LIN {X 0,Y 309.388,Z 528.778,A -85,B 0,C 180,E1 -16861.301,E2 -16861.301} C_VEL
LIN {X 0,Y 303.998,Z 522.37,A -85,B 0,C 180,E1 -16862.326,E2 -16862.326} C_VEL
LIN {X 0,Y 299.975,Z 517.415,A -85,B 0,C 180,E1 -16863.035,E2 -16863.035} C_VEL
LIN {X 0,Y 294.271,Z 509.19,A -85,B 0,C 180,E1 -16864.039,E2 -16864.039} C_VEL
LIN {X 0,Y 291.63,Z 504.474,A -85,B 0,C 180,E1 -16864.56,E2 -16864.56} C_VEL
LIN {X 0,Y 291.395,Z 503.436,A -85,B 0,C 180,E1 -16864.862,E2 -16864.862} C_VEL
LIN {X 0,Y 291.393,Z 503.278,A -85,B 0,C 180,E1 -16867.26,E2 -16867.26} C_VEL
LIN {X 0,Y 291.4,Z 503.295,A -85,B 0,C 180,E1 -16870.63,E2 -16870.63} C_VEL
LIN {X 0,Y 291.4,Z 503.269,A -85,B 0,C 180,E1 -16874.379,E2 -16874.379} C_VEL
LIN {X 0,Y 291.383,Z 503.302,A -85,B 0,C 180,E1 -16878.39,E2 -16878.39} C_VEL
LIN {X 0,Y 291.377,Z 503.316,A -85,B 0,C 180,E1 -16881.163,E2 -16881.163} C_VEL
LIN {X 0,Y 291.378,Z 503.299,A -85,B 0,C 180,E1 -16884.629,E2 -16884.629} C_VEL
LIN {X 0,Y 291.368,Z 503.305,A -85,B 0,C 180,E1 -16887.951,E2 -16887.951} C_VEL
LIN {X 0,Y 291.376,Z 503.307,A -85,B 0,C 180,E1 -16891.159,E2 -16891.159} C_VEL
LIN {X 0,Y 291.409,Z 503.295,A -85,B 0,C 180,E1 -16894.272,E2 -16894.272} C_VEL
LIN {X 0,Y 291.374,Z 503.303,A -85,B 0,C 180,E1 -16897.3,E2 -16897.3} C_VEL
LIN {X 0,Y 291.451,Z 503.298,A -85,B 0,C 180,E1 -16900.27,E2 -16900.27} C_VEL
LIN {X 0,Y 291.534,Z 503.284,A -85,B 0,C 180,E1 -16904.635,E2 -16904.635} C_VEL
LIN {X 0,Y 291.528,Z 503.272,A -85,B 0,C 180,E1 -16908.881,E2 -16908.881} C_VEL
LIN {X 0,Y 291.681,Z 503.258,A -85,B 0,C 180,E1 -16911.688,E2 -16911.688} C_VEL
LIN {X 0,Y 291.623,Z 503.281,A -85,B 0,C 180,E1 -16914.469,E2 -16914.469} C_VEL
LIN {X 0,Y 291.883,Z 503.219,A -85,B 0,C 180,E1 -16918.621,E2 -16918.621} C_VEL
LIN {X 0,Y 291.883,Z 503.248,A -85,B 0,C 180,E1 -16921.38,E2 -16921.38} C_VEL
LIN {X 0,Y 291.736,Z 503.243,A -85,B 0,C 180,E1 -16926.919,E2 -16926.919} C_VEL
LIN {X 0,Y 291.623,Z 503.283,A -85,B 0,C 180,E1 -16929.713,E2 -16929.713} C_VEL
LIN {X 0,Y 291.511,Z 503.266,A -85,B 0,C 180,E1 -16933.881,E2 -16933.881} C_VEL
LIN {X 0,Y 290.876,Z 503.358,A -85,B 0,C 180,E1 -16935.034,E2 -16935.034} C_VEL
LIN {X 0,Y 287.966,Z 503.74,A -85,B 0,C 180,E1 -16936.908,E2 -16936.908} C_VEL
LIN {X 0,Y 285.486,Z 504.04,A -85,B 0,C 180,E1 -16938.43,E2 -16938.43} C_VEL
LIN {X 0,Y 284.448,Z 504.156,A -85,B 0,C 180,E1 -16939.612,E2 -16939.612} C_VEL
LIN {X 0,Y 284.379,Z 504.161,A -85,B 0,C 180,E1 -16940.012,E2 -16940.012} C_VEL
LIN {X 0,Y 284.33,Z 504.191,A -85,B 0,C 180,E1 -16943.86,E2 -16943.86} C_VEL
LIN {X 0,Y 284.388,Z 504.161,A -85,B 0,C 180,E1 -16947.172,E2 -16947.172} C_VEL
LIN {X 0,Y 284.29,Z 504.193,A -85,B 0,C 180,E1 -16951.276,E2 -16951.276} C_VEL
LIN {X 0,Y 284.359,Z 504.19,A -85,B 0,C 180,E1 -16955.355,E2 -16955.355} C_VEL
LIN {X 0,Y 284.327,Z 504.179,A -85,B 0,C 180,E1 -16958.167,E2 -16958.167} C_VEL
LIN {X 0,Y 284.3,Z 504.187,A -85,B 0,C 180,E1 -16961.871,E2 -16961.871} C_VEL
LIN {X 0,Y 284.253,Z 504.171,A -85,B 0,C 180,E1 -16966.19,E2 -16966.19} C_VEL
LIN {X 0,Y 284.335,Z 504.299,A -85,B 0,C 180,E1 -16968.964,E2 -16968.964} C_VEL
LIN {X 0,Y 286.321,Z 512.531,A -85,B 0,C 180,E1 -16972.592,E2 -16972.592} C_VEL
LIN {X 0,Y 287.571,Z 518.102,A -85,B 0,C 180,E1 -16974.858,E2 -16974.858} C_VEL
LIN {X 0,Y 290.631,Z 524.68,A -85,B 0,C 180,E1 -16975.534,E2 -16975.534} C_VEL
LIN {X 0,Y 297.502,Z 539.552,A -85,B 0,C 180,E1 -16976.851,E2 -16976.851} C_VEL
LIN {X 0,Y 300.601,Z 547.16,A -85,B 0,C 180,E1 -16977.444,E2 -16977.444} C_VEL
LIN {X 0,Y 304.86,Z 568.834,A -85,B 0,C 180,E1 -16978.537,E2 -16978.537} C_VEL
LIN {X 0,Y 305.547,Z 572.651,A -85,B 0,C 180,E1 -16978.718,E2 -16978.718} C_VEL
LIN {X 0,Y 302.81,Z 652.99,A -85,B 0,C 180,E1 -16980.599,E2 -16980.599} C_VEL
LIN {X 0,Y 302.066,Z 664.113,A -85,B 0,C 180,E1 -16980.991,E2 -16980.991} C_VEL
LIN {X 0,Y 301.043,Z 674.654,A -85,B 0,C 180,E1 -16981.503,E2 -16981.503} C_VEL
LIN {X 0,Y 299.622,Z 685.804,A -85,B 0,C 180,E1 -16982.213,E2 -16982.213} C_VEL
LIN {X 0,Y 298.202,Z 695.774,A -85,B 0,C 180,E1 -16983.021,E2 -16983.021} C_VEL
LIN {X 0,Y 296.541,Z 705.698,A -85,B 0,C 180,E1 -16983.996,E2 -16983.996} C_VEL
LIN {X 0,Y 294.822,Z 715.628,A -85,B 0,C 180,E1 -16985.189,E2 -16985.189} C_VEL
LIN {X 0,Y 292.991,Z 724.837,A -85,B 0,C 180,E1 -16986.498,E2 -16986.498} C_VEL
LIN {X 0,Y 290.978,Z 733.855,A -85,B 0,C 180,E1 -16988.015,E2 -16988.015} C_VEL
LIN {X 0,Y 289.468,Z 740.831,A -85,B 0,C 180,E1 -16989.388,E2 -16989.388} C_VEL
LIN {X 0,Y 287.783,Z 748.355,A -85,B 0,C 180,E1 -16991.121,E2 -16991.121} C_VEL
LIN {X 0,Y 286.364,Z 754.83,A -85,B 0,C 180,E1 -16992.872,E2 -16992.872} C_VEL
LIN {X 0,Y 285.058,Z 761.375,A -85,B 0,C 180,E1 -16994.997,E2 -16994.997} C_VEL
LIN {X 0,Y 283.97,Z 766.81,A -85,B 0,C 180,E1 -16997.13,E2 -16997.13} C_VEL
LIN {X 0,Y 283.149,Z 771.256,A -85,B 0,C 180,E1 -16999.272,E2 -16999.272} C_VEL
LIN {X 0,Y 282.689,Z 774.805,A -85,B 0,C 180,E1 -17001.422,E2 -17001.422} C_VEL
LIN {X 0,Y 282.492,Z 776.748,A -85,B 0,C 180,E1 -17002.854,E2 -17002.854} C_VEL
LIN {X 0,Y 282.301,Z 779.436,A -85,B 0,C 180,E1 -17005.717,E2 -17005.717} C_VEL
LIN {X 0,Y 282.333,Z 780.256,A -85,B 0,C 180,E1 -17007.146,E2 -17007.146} C_VEL
LIN {X 0,Y 282.356,Z 780.984,A -85,B 0,C 180,E1 -17010,E2 -17010} C_VEL
LIN {X 0,Y 282.333,Z 780.256,A -85,B 0,C 180,E1 -17012.854,E2 -17012.854} C_VEL
LIN {X 0,Y 282.355,Z 778.546,A -85,B 0,C 180,E1 -17015.357,E2 -17015.357} C_VEL
LIN {X 0,Y 282.492,Z 776.748,A -85,B 0,C 180,E1 -17017.146,E2 -17017.146} C_VEL
LIN {X 0,Y 282.84,Z 773.788,A -85,B 0,C 180,E1 -17019.294,E2 -17019.294} C_VEL
LIN {X 0,Y 283.347,Z 769.956,A -85,B 0,C 180,E1 -17021.445,E2 -17021.445} C_VEL
LIN {X 0,Y 284.308,Z 765.194,A -85,B 0,C 180,E1 -17023.582,E2 -17023.582} C_VEL
LIN {X 0,Y 285.716,Z 757.793,A -85,B 0,C 180,E1 -17026.21,E2 -17026.21} C_VEL
LIN {X 0,Y 287.184,Z 751.03,A -85,B 0,C 180,E1 -17028.181,E2 -17028.181} C_VEL
LIN {X 0,Y 288.771,Z 743.955,A -85,B 0,C 180,E1 -17029.921,E2 -17029.921} C_VEL
LIN {X 0,Y 290.563,Z 735.674,A -85,B 0,C 180,E1 -17031.645,E2 -17031.645} C_VEL
LIN {X 0,Y 292.559,Z 726.957,A -85,B 0,C 180,E1 -17033.164,E2 -17033.164} C_VEL
LIN {X 0,Y 294.397,Z 718.265,A -85,B 0,C 180,E1 -17034.45,E2 -17034.45} C_VEL
LIN {X 0,Y 296.029,Z 708.918,A -85,B 0,C 180,E1 -17035.637,E2 -17035.637} C_VEL
LIN {X 0,Y 297.651,Z 699.282,A -85,B 0,C 180,E1 -17036.654,E2 -17036.654} C_VEL
LIN {X 0,Y 299.14,Z 689.023,A -85,B 0,C 180,E1 -17037.55,E2 -17037.55} C_VEL
LIN {X 0,Y 300.711,Z 677.373,A -85,B 0,C 180,E1 -17038.341,E2 -17038.341} C_VEL
LIN {X 0,Y 301.886,Z 665.937,A -85,B 0,C 180,E1 -17038.933,E2 -17038.933} C_VEL
LIN {X 0,Y 302.666,Z 655.532,A -85,B 0,C 180,E1 -17039.323,E2 -17039.323} C_VEL
LIN {X 0,Y 303.874,Z 624.474,A -85,B 0,C 180,E1 -17040.079,E2 -17040.079} C_VEL
LIN {X 0,Y 305.503,Z 572.378,A -85,B 0,C 180,E1 -17041.295,E2 -17041.295} C_VEL
LIN {X 0,Y 301.116,Z 549.474,A -85,B 0,C 180,E1 -17042.43,E2 -17042.43} C_VEL
LIN {X 0,Y 299.906,Z 545.142,A -85,B 0,C 180,E1 -17042.696,E2 -17042.696} C_VEL
LIN {X 0,Y 292.856,Z 529.335,A -85,B 0,C 180,E1 -17044.035,E2 -17044.035} C_VEL
LIN {X 0,Y 288.905,Z 521.195,A -85,B 0,C 180,E1 -17044.803,E2 -17044.803} C_VEL
LIN {X 0,Y 287.579,Z 518.084,A -85,B 0,C 180,E1 -17045.142,E2 -17045.142} C_VEL
LIN {X 0,Y 285.919,Z 510.842,A -85,B 0,C 180,E1 -17048.133,E2 -17048.133} C_VEL
LIN {X 0,Y 284.308,Z 504.269,A -85,B 0,C 180,E1 -17051.099,E2 -17051.099} C_VEL
LIN {X 0,Y 284.243,Z 504.173,A -85,B 0,C 180,E1 -17054.189,E2 -17054.189} C_VEL
LIN {X 0,Y 284.3,Z 504.186,A -85,B 0,C 180,E1 -17058.129,E2 -17058.129} C_VEL
LIN {X 0,Y 284.327,Z 504.179,A -85,B 0,C 180,E1 -17061.833,E2 -17061.833} C_VEL
LIN {X 0,Y 284.321,Z 504.186,A -85,B 0,C 180,E1 -17065.352,E2 -17065.352} C_VEL
LIN {X 0,Y 284.29,Z 504.193,A -85,B 0,C 180,E1 -17068.724,E2 -17068.724} C_VEL
LIN {X 0,Y 284.388,Z 504.161,A -85,B 0,C 180,E1 -17072.828,E2 -17072.828} C_VEL
LIN {X 0,Y 284.329,Z 504.192,A -85,B 0,C 180,E1 -17076.703,E2 -17076.703} C_VEL
LIN {X 0,Y 284.394,Z 504.173,A -85,B 0,C 180,E1 -17081.26,E2 -17081.26} C_VEL
LIN {X 0,Y 284.473,Z 504.163,A -85,B 0,C 180,E1 -17084.469,E2 -17084.469} C_VEL
LIN {X 0,Y 284.482,Z 504.164,A -85,B 0,C 180,E1 -17088.601,E2 -17088.601} C_VEL
LIN {X 0,Y 284.651,Z 504.146,A -85,B 0,C 180,E1 -17091.48,E2 -17091.48} C_VEL
LIN {X 0,Y 284.593,Z 504.124,A -85,B 0,C 180,E1 -17094.33,E2 -17094.33} C_VEL
LIN {X 0,Y 284.849,Z 504.124,A -85,B 0,C 180,E1 -17098.586,E2 -17098.586} C_VEL
LIN {X 0,Y 284.849,Z 504.094,A -85,B 0,C 180,E1 -17101.413,E2 -17101.413} C_VEL
LIN {X 0,Y 284.68,Z 504.143,A -85,B 0,C 180,E1 -17107.09,E2 -17107.09} C_VEL
LIN {X 0,Y 284.512,Z 504.137,A -85,B 0,C 180,E1 -17109.957,E2 -17109.957} C_VEL
LIN {X 0,Y 284.471,Z 504.173,A -85,B 0,C 180,E1 -17114.303,E2 -17114.303} C_VEL
LIN {X 0,Y 284.418,Z 504.152,A -85,B 0,C 180,E1 -17117.248,E2 -17117.248} C_VEL
LIN {X 0,Y 284.372,Z 504.187,A -85,B 0,C 180,E1 -17120.242,E2 -17120.242} C_VEL
LIN {X 0,Y 284.362,Z 504.163,A -85,B 0,C 180,E1 -17123.875,E2 -17123.875} C_VEL
LIN {X 0,Y 284.391,Z 504.184,A -85,B 0,C 180,E1 -17127.173,E2 -17127.173} C_VEL
LIN {X 0,Y 284.291,Z 504.177,A -85,B 0,C 180,E1 -17131.274,E2 -17131.274} C_VEL
LIN {X 0,Y 284.355,Z 504.174,A -85,B 0,C 180,E1 -17135.354,E2 -17135.354} C_VEL
LIN {X 0,Y 284.328,Z 504.195,A -85,B 0,C 180,E1 -17138.165,E2 -17138.165} C_VEL
LIN {X 0,Y 284.337,Z 504.186,A -85,B 0,C 180,E1 -17142.141,E2 -17142.141} C_VEL
LIN {X 0,Y 284.346,Z 504.141,A -85,B 0,C 180,E1 -17146.208,E2 -17146.208} C_VEL
LIN {X 0,Y 284.346,Z 504.19,A -85,B 0,C 180,E1 -17150.013,E2 -17150.013} C_VEL
LIN {X 0,Y 284.359,Z 504.268,A -85,B 0,C 180,E1 -17154.145,E2 -17154.145} C_VEL
LIN {X 0,Y 284.53,Z 505.129,A -85,B 0,C 180,E1 -17154.453,E2 -17154.453} C_VEL
LIN {X 0,Y 286.104,Z 508.057,A -85,B 0,C 180,E1 -17154.806,E2 -17154.806} C_VEL
LIN {X 0,Y 293.317,Z 519.531,A -85,B 0,C 180,E1 -17156.134,E2 -17156.134} C_VEL
LIN {X 0,Y 299.003,Z 526.765,A -85,B 0,C 180,E1 -17157.104,E2 -17157.104} C_VEL
LIN {X 0,Y 304.272,Z 532.807,A -85,B 0,C 180,E1 -17158.034,E2 -17158.034} C_VEL
LIN {X 0,Y 309.399,Z 538.457,A -85,B 0,C 180,E1 -17158.999,E2 -17158.999} C_VEL
LIN {X 0,Y 317.099,Z 546.681,A -85,B 0,C 180,E1 -17160.597,E2 -17160.597} C_VEL
LIN {X 0,Y 324.724,Z 554.633,A -85,B 0,C 180,E1 -17162.359,E2 -17162.359} C_VEL
LIN {X 0,Y 330.496,Z 560.265,A -85,B 0,C 180,E1 -17163.781,E2 -17163.781} C_VEL
LIN {X 0,Y 338.132,Z 567.499,A -85,B 0,C 180,E1 -17165.784,E2 -17165.784} C_VEL
LIN {X 0,Y 345.106,Z 573.723,A -85,B 0,C 180,E1 -17167.758,E2 -17167.758} C_VEL
LIN {X 0,Y 349.979,Z 577.935,A -85,B 0,C 180,E1 -17169.237,E2 -17169.237} C_VEL
LIN {X 0,Y 352.665,Z 580.136,A -85,B 0,C 180,E1 -17170.097,E2 -17170.097} C_VEL
LIN {X 0,Y 357.635,Z 584.572,A -85,B 0,C 180,E1 -17171.813,E2 -17171.813} C_VEL
LIN {X 0,Y 361.888,Z 587.705,A -85,B 0,C 180,E1 -17173.392,E2 -17173.392} C_VEL
LIN {X 0,Y 365.95,Z 591.436,A -85,B 0,C 180,E1 -17175.092,E2 -17175.092} C_VEL
LIN {X 0,Y 369.976,Z 594.165,A -85,B 0,C 180,E1 -17176.93,E2 -17176.93} C_VEL
LIN {X 0,Y 372.105,Z 595.489,A -85,B 0,C 180,E1 -17178.009,E2 -17178.009} C_VEL
LIN {X 0,Y 375.607,Z 598.813,A -85,B 0,C 180,E1 -17180.125,E2 -17180.125} C_VEL
LIN {X 0,Y 378.307,Z 600.726,A -85,B 0,C 180,E1 -17182.068,E2 -17182.068} C_VEL
LIN {X 0,Y 380.59,Z 602.028,A -85,B 0,C 180,E1 -17184.161,E2 -17184.161} C_VEL
LIN {X 0,Y 381.878,Z 602.601,A -85,B 0,C 180,E1 -17185.778,E2 -17185.778} C_VEL
LIN {X 0,Y 382.982,Z 603.01,A -85,B 0,C 180,E1 -17187.897,E2 -17187.897} C_VEL
LIN {X 0,Y 383.245,Z 603.22,A -85,B 0,C 180,E1 -17188.949,E2 -17188.949} C_VEL
LIN {X 0,Y 383.354,Z 603.112,A -85,B 0,C 180,E1 -17190,E2 -17190} C_VEL
LIN {X 0,Y 383.122,Z 603.129,A -85,B 0,C 180,E1 -17191.577,E2 -17191.577} C_VEL
LIN {X 0,Y 382.533,Z 602.752,A -85,B 0,C 180,E1 -17193.159,E2 -17193.159} C_VEL
LIN {X 0,Y 381.067,Z 602.238,A -85,B 0,C 180,E1 -17195.291,E2 -17195.291} C_VEL
LIN {X 0,Y 378.865,Z 601.078,A -85,B 0,C 180,E1 -17197.461,E2 -17197.461} C_VEL
LIN {X 0,Y 376.03,Z 599.118,A -85,B 0,C 180,E1 -17199.595,E2 -17199.595} C_VEL
LIN {X 0,Y 372.797,Z 596.178,A -85,B 0,C 180,E1 -17201.605,E2 -17201.605} C_VEL
LIN {X 0,Y 370.828,Z 594.6,A -85,B 0,C 180,E1 -17202.657,E2 -17202.657} C_VEL
LIN {X 0,Y 366.877,Z 592.133,A -85,B 0,C 180,E1 -17204.51,E2 -17204.51} C_VEL
LIN {X 0,Y 362.424,Z 588.26,A -85,B 0,C 180,E1 -17206.396,E2 -17206.396} C_VEL
LIN {X 0,Y 360.069,Z 586.255,A -85,B 0,C 180,E1 -17207.309,E2 -17207.309} C_VEL
LIN {X 0,Y 355.388,Z 582.701,A -85,B 0,C 180,E1 -17208.978,E2 -17208.978} C_VEL
LIN {X 0,Y 350.833,Z 578.603,A -85,B 0,C 180,E1 -17210.49,E2 -17210.49} C_VEL
LIN {X 0,Y 345.814,Z 574.415,A -85,B 0,C 180,E1 -17212.027,E2 -17212.027} C_VEL
LIN {X 0,Y 341.845,Z 570.783,A -85,B 0,C 180,E1 -17213.188,E2 -17213.188} C_VEL
LIN {X 0,Y 336.549,Z 565.919,A -85,B 0,C 180,E1 -17214.645,E2 -17214.645} C_VEL
LIN {X 0,Y 329.814,Z 559.585,A -85,B 0,C 180,E1 -17216.389,E2 -17216.389} C_VEL
LIN {X 0,Y 322.602,Z 552.32,A -85,B 0,C 180,E1 -17218.156,E2 -17218.156} C_VEL
LIN {X 0,Y 316.361,Z 545.833,A -85,B 0,C 180,E1 -17219.571,E2 -17219.571} C_VEL
LIN {X 0,Y 308.074,Z 537.151,A -85,B 0,C 180,E1 -17221.258,E2 -17221.258} C_VEL
LIN {X 0,Y 300.15,Z 528.128,A -85,B 0,C 180,E1 -17222.705,E2 -17222.705} C_VEL
LIN {X 0,Y 295.167,Z 521.883,A -85,B 0,C 180,E1 -17223.556,E2 -17223.556} C_VEL
LIN {X 0,Y 289.497,Z 513.766,A -85,B 0,C 180,E1 -17224.549,E2 -17224.549} C_VEL
LIN {X 0,Y 285.82,Z 507.682,A -85,B 0,C 180,E1 -17225.245,E2 -17225.245} C_VEL
LIN {X 0,Y 284.493,Z 505.002,A -85,B 0,C 180,E1 -17225.575,E2 -17225.575} C_VEL
LIN {X 0,Y 284.335,Z 504.221,A -85,B 0,C 180,E1 -17225.949,E2 -17225.949} C_VEL
LIN {X 0,Y 284.346,Z 504.19,A -85,B 0,C 180,E1 -17229.987,E2 -17229.987} C_VEL
LIN {X 0,Y 284.349,Z 504.144,A -85,B 0,C 180,E1 -17234.213,E2 -17234.213} C_VEL
LIN {X 0,Y 284.334,Z 504.182,A -85,B 0,C 180,E1 -17238.137,E2 -17238.137} C_VEL
LIN {X 0,Y 284.336,Z 504.188,A -85,B 0,C 180,E1 -17242.273,E2 -17242.273} C_VEL
LIN {X 0,Y 284.317,Z 504.186,A -85,B 0,C 180,E1 -17245.353,E2 -17245.353} C_VEL
LIN {X 0,Y 284.291,Z 504.177,A -85,B 0,C 180,E1 -17248.726,E2 -17248.726} C_VEL
LIN {X 0,Y 284.391,Z 504.184,A -85,B 0,C 180,E1 -17252.827,E2 -17252.827} C_VEL
LIN {X 0,Y 284.359,Z 504.167,A -85,B 0,C 180,E1 -17256.707,E2 -17256.707} C_VEL
LIN {X 0,Y 284.396,Z 504.164,A -85,B 0,C 180,E1 -17261.262,E2 -17261.262} C_VEL
LIN {X 0,Y 284.471,Z 504.161,A -85,B 0,C 180,E1 -17264.47,E2 -17264.47} C_VEL
LIN {X 0,Y 284.48,Z 504.153,A -85,B 0,C 180,E1 -17268.602,E2 -17268.602} C_VEL
LIN {X 0,Y 284.632,Z 504.131,A -85,B 0,C 180,E1 -17271.481,E2 -17271.481} C_VEL
LIN {X 0,Y 284.593,Z 504.158,A -85,B 0,C 180,E1 -17274.332,E2 -17274.332} C_VEL
LIN {X 0,Y 284.849,Z 504.094,A -85,B 0,C 180,E1 -17278.587,E2 -17278.587} C_VEL
LIN {X 0,Y 284.849,Z 504.124,A -85,B 0,C 180,E1 -17281.414,E2 -17281.414} C_VEL
LIN {X 0,Y 284.688,Z 504.122,A -85,B 0,C 180,E1 -17287.091,E2 -17287.091} C_VEL
LIN {X 0,Y 284.561,Z 504.164,A -85,B 0,C 180,E1 -17289.956,E2 -17289.956} C_VEL
LIN {X 0,Y 284.472,Z 504.145,A -85,B 0,C 180,E1 -17294.304,E2 -17294.304} C_VEL
LIN {X 0,Y 284.418,Z 504.181,A -85,B 0,C 180,E1 -17297.249,E2 -17297.249} C_VEL
LIN {X 0,Y 284.379,Z 504.161,A -85,B 0,C 180,E1 -17300.012,E2 -17300.012} C_VEL
LIN {X 0,Y 283.742,Z 504.243,A -85,B 0,C 180,E1 -17301.195,E2 -17301.195} C_VEL
LIN {X 0,Y 280.862,Z 504.62,A -85,B 0,C 180,E1 -17303.12,E2 -17303.12} C_VEL
LIN {X 0,Y 278.406,Z 504.928,A -85,B 0,C 180,E1 -17304.683,E2 -17304.683} C_VEL
LIN {X 0,Y 277.371,Z 505.044,A -85,B 0,C 180,E1 -17305.896,E2 -17305.896} C_VEL
LIN {X 0,Y 277.298,Z 505.047,A -85,B 0,C 180,E1 -17306.307,E2 -17306.307} C_VEL
LIN {X 0,Y 277.269,Z 505.074,A -85,B 0,C 180,E1 -17310.482,E2 -17310.482} C_VEL
LIN {X 0,Y 277.251,Z 505.057,A -85,B 0,C 180,E1 -17313.896,E2 -17313.896} C_VEL
LIN {X 0,Y 277.282,Z 505.057,A -85,B 0,C 180,E1 -17317.468,E2 -17317.468} C_VEL
LIN {X 0,Y 277.238,Z 505.069,A -85,B 0,C 180,E1 -17321.232,E2 -17321.232} C_VEL
LIN {X 0,Y 277.202,Z 505.059,A -85,B 0,C 180,E1 -17325.227,E2 -17325.227} C_VEL
LIN {X 0,Y 277.252,Z 505.202,A -85,B 0,C 180,E1 -17328.181,E2 -17328.181} C_VEL
LIN {X 0,Y 278.955,Z 512.096,A -85,B 0,C 180,E1 -17331.354,E2 -17331.354} C_VEL
LIN {X 0,Y 280.3,Z 517.888,A -85,B 0,C 180,E1 -17333.811,E2 -17333.811} C_VEL
LIN {X 0,Y 283.792,Z 525.156,A -85,B 0,C 180,E1 -17334.602,E2 -17334.602} C_VEL
LIN {X 0,Y 291.131,Z 540.673,A -85,B 0,C 180,E1 -17336.067,E2 -17336.067} C_VEL
LIN {X 0,Y 294.935,Z 550.002,A -85,B 0,C 180,E1 -17336.825,E2 -17336.825} C_VEL
LIN {X 0,Y 299.104,Z 571.908,A -85,B 0,C 180,E1 -17337.95,E2 -17337.95} C_VEL
LIN {X 0,Y 299.446,Z 574.809,A -85,B 0,C 180,E1 -17338.071,E2 -17338.071} C_VEL
LIN {X 0,Y 296.651,Z 652.969,A -85,B 0,C 180,E1 -17339.933,E2 -17339.933} C_VEL
LIN {X 0,Y 295.876,Z 663.915,A -85,B 0,C 180,E1 -17340.324,E2 -17340.324} C_VEL
LIN {X 0,Y 294.834,Z 674.457,A -85,B 0,C 180,E1 -17340.846,E2 -17340.846} C_VEL
LIN {X 0,Y 293.349,Z 685.606,A -85,B 0,C 180,E1 -17341.566,E2 -17341.566} C_VEL
LIN {X 0,Y 291.888,Z 695.576,A -85,B 0,C 180,E1 -17342.388,E2 -17342.388} C_VEL
LIN {X 0,Y 290.159,Z 705.494,A -85,B 0,C 180,E1 -17343.379,E2 -17343.379} C_VEL
LIN {X 0,Y 288.566,Z 714.474,A -85,B 0,C 180,E1 -17344.464,E2 -17344.464} C_VEL
LIN {X 0,Y 286.488,Z 724.639,A -85,B 0,C 180,E1 -17345.932,E2 -17345.932} C_VEL
LIN {X 0,Y 284.363,Z 733.656,A -85,B 0,C 180,E1 -17347.476,E2 -17347.476} C_VEL
LIN {X 0,Y 282.803,Z 740.632,A -85,B 0,C 180,E1 -17348.879,E2 -17348.879} C_VEL
LIN {X 0,Y 281.037,Z 748.155,A -85,B 0,C 180,E1 -17350.65,E2 -17350.65} C_VEL
LIN {X 0,Y 279.535,Z 754.631,A -85,B 0,C 180,E1 -17352.441,E2 -17352.441} C_VEL
LIN {X 0,Y 278.165,Z 761.176,A -85,B 0,C 180,E1 -17354.616,E2 -17354.616} C_VEL
LIN {X 0,Y 276.994,Z 766.61,A -85,B 0,C 180,E1 -17356.8,E2 -17356.8} C_VEL
LIN {X 0,Y 276.133,Z 771.057,A -85,B 0,C 180,E1 -17358.996,E2 -17358.996} C_VEL
LIN {X 0,Y 275.641,Z 774.606,A -85,B 0,C 180,E1 -17361.2,E2 -17361.2} C_VEL
LIN {X 0,Y 275.42,Z 776.549,A -85,B 0,C 180,E1 -17362.67,E2 -17362.67} C_VEL
LIN {X 0,Y 275.216,Z 779.238,A -85,B 0,C 180,E1 -17365.606,E2 -17365.606} C_VEL
LIN {X 0,Y 275.26,Z 780.533,A -85,B 0,C 180,E1 -17368.537,E2 -17368.537} C_VEL
LIN {X 0,Y 275.278,Z 780.786,A -85,B 0,C 180,E1 -17370,E2 -17370} C_VEL
LIN {X 0,Y 275.242,Z 780.058,A -85,B 0,C 180,E1 -17372.927,E2 -17372.927} C_VEL
LIN {X 0,Y 275.246,Z 778.583,A -85,B 0,C 180,E1 -17375.243,E2 -17375.243} C_VEL
LIN {X 0,Y 275.42,Z 776.549,A -85,B 0,C 180,E1 -17377.33,E2 -17377.33} C_VEL
LIN {X 0,Y 275.794,Z 773.589,A -85,B 0,C 180,E1 -17379.534,E2 -17379.534} C_VEL
LIN {X 0,Y 276.343,Z 769.757,A -85,B 0,C 180,E1 -17381.739,E2 -17381.739} C_VEL
LIN {X 0,Y 277.359,Z 764.994,A -85,B 0,C 180,E1 -17383.929,E2 -17383.929} C_VEL
LIN {X 0,Y 278.584,Z 759.185,A -85,B 0,C 180,E1 -17386.111,E2 -17386.111} C_VEL
LIN {X 0,Y 280.092,Z 752.169,A -85,B 0,C 180,E1 -17388.279,E2 -17388.279} C_VEL
LIN {X 0,Y 282.063,Z 743.756,A -85,B 0,C 180,E1 -17390.415,E2 -17390.415} C_VEL
LIN {X 0,Y 283.511,Z 737.292,A -85,B 0,C 180,E1 -17391.828,E2 -17391.828} C_VEL
LIN {X 0,Y 285.785,Z 727.818,A -85,B 0,C 180,E1 -17393.554,E2 -17393.554} C_VEL
LIN {X 0,Y 287.864,Z 718.395,A -85,B 0,C 180,E1 -17394.992,E2 -17394.992} C_VEL
LIN {X 0,Y 289.403,Z 709.888,A -85,B 0,C 180,E1 -17396.113,E2 -17396.113} C_VEL
LIN {X 0,Y 291.307,Z 699.083,A -85,B 0,C 180,E1 -17397.283,E2 -17397.283} C_VEL
LIN {X 0,Y 292.87,Z 688.825,A -85,B 0,C 180,E1 -17398.192,E2 -17398.192} C_VEL
LIN {X 0,Y 294.472,Z 677.175,A -85,B 0,C 180,E1 -17398.998,E2 -17398.998} C_VEL
LIN {X 0,Y 295.69,Z 665.739,A -85,B 0,C 180,E1 -17399.599,E2 -17399.599} C_VEL
LIN {X 0,Y 296.494,Z 655.438,A -85,B 0,C 180,E1 -17399.992,E2 -17399.992} C_VEL
LIN {X 0,Y 297.797,Z 623.575,A -85,B 0,C 180,E1 -17400.778,E2 -17400.778} C_VEL
LIN {X 0,Y 299.362,Z 573.447,A -85,B 0,C 180,E1 -17401.977,E2 -17401.977} C_VEL
LIN {X 0,Y 295.766,Z 553.886,A -85,B 0,C 180,E1 -17402.961,E2 -17402.961} C_VEL
LIN {X 0,Y 294.32,Z 548.2,A -85,B 0,C 180,E1 -17403.304,E2 -17403.304} C_VEL
LIN {X 0,Y 287.542,Z 532.922,A -85,B 0,C 180,E1 -17404.642,E2 -17404.642} C_VEL
LIN {X 0,Y 281.806,Z 521.217,A -85,B 0,C 180,E1 -17405.804,E2 -17405.804} C_VEL
LIN {X 0,Y 280.279,Z 517.738,A -85,B 0,C 180,E1 -17406.223,E2 -17406.223} C_VEL
LIN {X 0,Y 278.315,Z 509.37,A -85,B 0,C 180,E1 -17409.869,E2 -17409.869} C_VEL
LIN {X 0,Y 277.254,Z 505.153,A -85,B 0,C 180,E1 -17411.886,E2 -17411.886} C_VEL
LIN {X 0,Y 277.206,Z 505.065,A -85,B 0,C 180,E1 -17415.224,E2 -17415.224} C_VEL
LIN {X 0,Y 277.285,Z 505.069,A -85,B 0,C 180,E1 -17419.495,E2 -17419.495} C_VEL
LIN {X 0,Y 277.282,Z 505.057,A -85,B 0,C 180,E1 -17422.532,E2 -17422.532} C_VEL
LIN {X 0,Y 277.251,Z 505.057,A -85,B 0,C 180,E1 -17426.104,E2 -17426.104} C_VEL
LIN {X 0,Y 277.258,Z 505.075,A -85,B 0,C 180,E1 -17429.538,E2 -17429.538} C_VEL
LIN {X 0,Y 277.35,Z 505.037,A -85,B 0,C 180,E1 -17432.862,E2 -17432.862} C_VEL
LIN {X 0,Y 277.292,Z 505.068,A -85,B 0,C 180,E1 -17436.076,E2 -17436.076} C_VEL
LIN {X 0,Y 277.338,Z 505.046,A -85,B 0,C 180,E1 -17440.765,E2 -17440.765} C_VEL
LIN {X 0,Y 277.423,Z 505.027,A -85,B 0,C 180,E1 -17445.325,E2 -17445.325} C_VEL
LIN {X 0,Y 277.501,Z 505.044,A -85,B 0,C 180,E1 -17449.788,E2 -17449.788} C_VEL
LIN {X 0,Y 277.644,Z 505.001,A -85,B 0,C 180,E1 -17452.728,E2 -17452.728} C_VEL
LIN {X 0,Y 277.815,Z 505,A -85,B 0,C 180,E1 -17458.55,E2 -17458.55} C_VEL
LIN {X 0,Y 277.815,Z 504.969,A -85,B 0,C 180,E1 -17461.449,E2 -17461.449} C_VEL
LIN {X 0,Y 277.634,Z 505.018,A -85,B 0,C 180,E1 -17467.271,E2 -17467.271} C_VEL
LIN {X 0,Y 277.454,Z 505.016,A -85,B 0,C 180,E1 -17470.212,E2 -17470.212} C_VEL
LIN {X 0,Y 277.421,Z 505.051,A -85,B 0,C 180,E1 -17474.674,E2 -17474.674} C_VEL
LIN {X 0,Y 277.338,Z 505.051,A -85,B 0,C 180,E1 -17479.234,E2 -17479.234} C_VEL
LIN {X 0,Y 277.312,Z 505.039,A -85,B 0,C 180,E1 -17484.17,E2 -17484.17} C_VEL
LIN {X 0,Y 277.32,Z 505.067,A -85,B 0,C 180,E1 -17487.505,E2 -17487.505} C_VEL
LIN {X 0,Y 277.266,Z 505.049,A -85,B 0,C 180,E1 -17490.481,E2 -17490.481} C_VEL
LIN {X 0,Y 277.248,Z 505.073,A -85,B 0,C 180,E1 -17493.895,E2 -17493.895} C_VEL
LIN {X 0,Y 277.281,Z 505.064,A -85,B 0,C 180,E1 -17497.466,E2 -17497.466} C_VEL
LIN {X 0,Y 277.259,Z 505.058,A -85,B 0,C 180,E1 -17501.226,E2 -17501.226} C_VEL
LIN {X 0,Y 277.282,Z 505.032,A -85,B 0,C 180,E1 -17505.208,E2 -17505.208} C_VEL
LIN {X 0,Y 277.29,Z 505.053,A -85,B 0,C 180,E1 -17509.495,E2 -17509.495} C_VEL
LIN {X 0,Y 277.32,Z 505.207,A -85,B 0,C 180,E1 -17513.147,E2 -17513.147} C_VEL
LIN {X 0,Y 277.534,Z 506.141,A -85,B 0,C 180,E1 -17513.45,E2 -17513.45} C_VEL
LIN {X 0,Y 279.182,Z 509.073,A -85,B 0,C 180,E1 -17513.823,E2 -17513.823} C_VEL
LIN {X 0,Y 288.794,Z 524.475,A -85,B 0,C 180,E1 -17515.672,E2 -17515.672} C_VEL
LIN {X 0,Y 294.96,Z 532.239,A -85,B 0,C 180,E1 -17516.714,E2 -17516.714} C_VEL
LIN {X 0,Y 303.207,Z 541.617,A -85,B 0,C 180,E1 -17518.135,E2 -17518.135} C_VEL
LIN {X 0,Y 311.733,Z 550.312,A -85,B 0,C 180,E1 -17519.753,E2 -17519.753} C_VEL
LIN {X 0,Y 317.673,Z 556.424,A -85,B 0,C 180,E1 -17521.016,E2 -17521.016} C_VEL
LIN {X 0,Y 324.213,Z 562.958,A -85,B 0,C 180,E1 -17522.532,E2 -17522.532} C_VEL
LIN {X 0,Y 331.515,Z 569.934,A -85,B 0,C 180,E1 -17524.343,E2 -17524.343} C_VEL
LIN {X 0,Y 338.931,Z 576.737,A -85,B 0,C 180,E1 -17526.313,E2 -17526.313} C_VEL
LIN {X 0,Y 342.658,Z 579.944,A -85,B 0,C 180,E1 -17527.361,E2 -17527.361} C_VEL
LIN {X 0,Y 347.773,Z 584.367,A -85,B 0,C 180,E1 -17528.886,E2 -17528.886} C_VEL
LIN {X 0,Y 351.33,Z 587.318,A -85,B 0,C 180,E1 -17530.006,E2 -17530.006} C_VEL
LIN {X 0,Y 356.653,Z 591.801,A -85,B 0,C 180,E1 -17531.817,E2 -17531.817} C_VEL
LIN {X 0,Y 360.423,Z 594.627,A -85,B 0,C 180,E1 -17533.206,E2 -17533.206} C_VEL
LIN {X 0,Y 364.739,Z 598.442,A -85,B 0,C 180,E1 -17534.979,E2 -17534.979} C_VEL
LIN {X 0,Y 368.744,Z 601.09,A -85,B 0,C 180,E1 -17536.779,E2 -17536.779} C_VEL
LIN {X 0,Y 370.987,Z 602.531,A -85,B 0,C 180,E1 -17537.904,E2 -17537.904} C_VEL
LIN {X 0,Y 374.535,Z 605.786,A -85,B 0,C 180,E1 -17540.009,E2 -17540.009} C_VEL
LIN {X 0,Y 377.137,Z 607.636,A -85,B 0,C 180,E1 -17541.84,E2 -17541.84} C_VEL
LIN {X 0,Y 379.705,Z 609.052,A -85,B 0,C 180,E1 -17544.147,E2 -17544.147} C_VEL
LIN {X 0,Y 381.001,Z 609.645,A -85,B 0,C 180,E1 -17545.769,E2 -17545.769} C_VEL
LIN {X 0,Y 382.115,Z 610.048,A -85,B 0,C 180,E1 -17547.892,E2 -17547.892} C_VEL
LIN {X 0,Y 382.38,Z 610.255,A -85,B 0,C 180,E1 -17548.947,E2 -17548.947} C_VEL
LIN {X 0,Y 382.489,Z 610.156,A -85,B 0,C 180,E1 -17550,E2 -17550} C_VEL
LIN {X 0,Y 382.253,Z 610.176,A -85,B 0,C 180,E1 -17551.58,E2 -17551.58} C_VEL
LIN {X 0,Y 381.661,Z 609.8,A -85,B 0,C 180,E1 -17553.167,E2 -17553.167} C_VEL
LIN {X 0,Y 380.18,Z 609.305,A -85,B 0,C 180,E1 -17555.303,E2 -17555.303} C_VEL
LIN {X 0,Y 377.958,Z 608.138,A -85,B 0,C 180,E1 -17557.479,E2 -17557.479} C_VEL
LIN {X 0,Y 375.232,Z 606.311,A -85,B 0,C 180,E1 -17559.527,E2 -17559.527} C_VEL
LIN {X 0,Y 372.197,Z 603.674,A -85,B 0,C 180,E1 -17561.423,E2 -17561.423} C_VEL
LIN {X 0,Y 369.835,Z 601.653,A -85,B 0,C 180,E1 -17562.692,E2 -17562.692} C_VEL
LIN {X 0,Y 365.831,Z 599.21,A -85,B 0,C 180,E1 -17564.552,E2 -17564.552} C_VEL
LIN {X 0,Y 361.481,Z 595.598,A -85,B 0,C 180,E1 -17566.379,E2 -17566.379} C_VEL
LIN {X 0,Y 358.562,Z 593.081,A -85,B 0,C 180,E1 -17567.5,E2 -17567.5} C_VEL
LIN {X 0,Y 353.762,Z 589.528,A -85,B 0,C 180,E1 -17569.18,E2 -17569.18} C_VEL
LIN {X 0,Y 349.079,Z 585.32,A -85,B 0,C 180,E1 -17570.72,E2 -17570.72} C_VEL
LIN {X 0,Y 343.664,Z 580.879,A -85,B 0,C 180,E1 -17572.35,E2 -17572.35} C_VEL
LIN {X 0,Y 339.332,Z 577.046,A -85,B 0,C 180,E1 -17573.579,E2 -17573.579} C_VEL
LIN {X 0,Y 333.706,Z 571.86,A -85,B 0,C 180,E1 -17575.098,E2 -17575.098} C_VEL
LIN {X 0,Y 327.189,Z 565.856,A -85,B 0,C 180,E1 -17576.746,E2 -17576.746} C_VEL
LIN {X 0,Y 319.729,Z 558.527,A -85,B 0,C 180,E1 -17578.52,E2 -17578.52} C_VEL
LIN {X 0,Y 313.159,Z 551.858,A -85,B 0,C 180,E1 -17579.946,E2 -17579.946} C_VEL
LIN {X 0,Y 304.653,Z 543.113,A -85,B 0,C 180,E1 -17581.602,E2 -17581.602} C_VEL
LIN {X 0,Y 296.252,Z 533.844,A -85,B 0,C 180,E1 -17583.067,E2 -17583.067} C_VEL
LIN {X 0,Y 290.549,Z 526.714,A -85,B 0,C 180,E1 -17584.025,E2 -17584.025} C_VEL
LIN {X 0,Y 284.719,Z 518.291,A -85,B 0,C 180,E1 -17585.082,E2 -17585.082} C_VEL
LIN {X 0,Y 279.012,Z 508.847,A -85,B 0,C 180,E1 -17586.21,E2 -17586.21} C_VEL
LIN {X 0,Y 277.527,Z 506.157,A -85,B 0,C 180,E1 -17586.548,E2 -17586.548} C_VEL
LIN {X 0,Y 277.309,Z 505.107,A -85,B 0,C 180,E1 -17586.91,E2 -17586.91} C_VEL
LIN {X 0,Y 277.26,Z 505.039,A -85,B 0,C 180,E1 -17591.226,E2 -17591.226} C_VEL
LIN {X 0,Y 277.282,Z 505.04,A -85,B 0,C 180,E1 -17595.208,E2 -17595.208} C_VEL
LIN {X 0,Y 277.289,Z 505.054,A -85,B 0,C 180,E1 -17599.494,E2 -17599.494} C_VEL
LIN {X 0,Y 277.281,Z 505.064,A -85,B 0,C 180,E1 -17602.534,E2 -17602.534} C_VEL
LIN {X 0,Y 277.248,Z 505.073,A -85,B 0,C 180,E1 -17606.105,E2 -17606.105} C_VEL
LIN {X 0,Y 277.255,Z 505.05,A -85,B 0,C 180,E1 -17609.539,E2 -17609.539} C_VEL
LIN {X 0,Y 277.352,Z 505.061,A -85,B 0,C 180,E1 -17612.864,E2 -17612.864} C_VEL
LIN {X 0,Y 277.321,Z 505.039,A -85,B 0,C 180,E1 -17616.08,E2 -17616.08} C_VEL
LIN {X 0,Y 277.338,Z 505.051,A -85,B 0,C 180,E1 -17620.766,E2 -17620.766} C_VEL
LIN {X 0,Y 277.421,Z 505.051,A -85,B 0,C 180,E1 -17625.326,E2 -17625.326} C_VEL
LIN {X 0,Y 277.454,Z 505.016,A -85,B 0,C 180,E1 -17629.788,E2 -17629.788} C_VEL
LIN {X 0,Y 277.635,Z 505.018,A -85,B 0,C 180,E1 -17632.729,E2 -17632.729} C_VEL
LIN {X 0,Y 277.815,Z 504.969,A -85,B 0,C 180,E1 -17638.551,E2 -17638.551} C_VEL
LIN {X 0,Y 277.815,Z 505,A -85,B 0,C 180,E1 -17641.45,E2 -17641.45} C_VEL
LIN {X 0,Y 277.644,Z 505.001,A -85,B 0,C 180,E1 -17647.272,E2 -17647.272} C_VEL
LIN {X 0,Y 277.501,Z 505.044,A -85,B 0,C 180,E1 -17650.212,E2 -17650.212} C_VEL
LIN {X 0,Y 277.423,Z 505.027,A -85,B 0,C 180,E1 -17654.675,E2 -17654.675} C_VEL
LIN {X 0,Y 277.338,Z 505.046,A -85,B 0,C 180,E1 -17659.235,E2 -17659.235} C_VEL
LIN {X 0,Y 277.287,Z 505.07,A -85,B 0,C 180,E1 -17664.158,E2 -17664.158} C_VEL
LIN {X 0,Y 277.298,Z 505.047,A -85,B 0,C 180,E1 -17666.307,E2 -17666.307} C_VEL
LIN {X 0,Y 276.64,Z 505.13,A -85,B 0,C 180,E1 -17667.519,E2 -17667.519} C_VEL
LIN {X 0,Y 273.725,Z 505.512,A -85,B 0,C 180,E1 -17669.492,E2 -17669.492} C_VEL
LIN {X 0,Y 271.261,Z 505.816,A -85,B 0,C 180,E1 -17671.095,E2 -17671.095} C_VEL
LIN {X 0,Y 270.239,Z 505.93,A -85,B 0,C 180,E1 -17672.339,E2 -17672.339} C_VEL
LIN {X 0,Y 270.177,Z 505.935,A -85,B 0,C 180,E1 -17672.761,E2 -17672.761} C_VEL
LIN {X 0,Y 270.238,Z 505.941,A -85,B 0,C 180,E1 -17676.739,E2 -17676.739} C_VEL
LIN {X 0,Y 270.235,Z 505.948,A -85,B 0,C 180,E1 -17680.556,E2 -17680.556} C_VEL
LIN {X 0,Y 270.157,Z 505.947,A -85,B 0,C 180,E1 -17684.62,E2 -17684.62} C_VEL
LIN {X 0,Y 270.209,Z 506.119,A -85,B 0,C 180,E1 -17687.365,E2 -17687.365} C_VEL
LIN {X 0,Y 272.163,Z 513.955,A -85,B 0,C 180,E1 -17691.103,E2 -17691.103} C_VEL
LIN {X 0,Y 273.078,Z 517.758,A -85,B 0,C 180,E1 -17692.714,E2 -17692.714} C_VEL
LIN {X 0,Y 275.146,Z 521.926,A -85,B 0,C 180,E1 -17693.219,E2 -17693.219} C_VEL
LIN {X 0,Y 282.333,Z 536.581,A -85,B 0,C 180,E1 -17694.741,E2 -17694.741} C_VEL
LIN {X 0,Y 289.104,Z 552.1,A -85,B 0,C 180,E1 -17696.133,E2 -17696.133} C_VEL
LIN {X 0,Y 293.173,Z 573.614,A -85,B 0,C 180,E1 -17697.275,E2 -17697.275} C_VEL
LIN {X 0,Y 293.412,Z 575.971,A -85,B 0,C 180,E1 -17697.372,E2 -17697.372} C_VEL
LIN {X 0,Y 290.515,Z 652.935,A -85,B 0,C 180,E1 -17699.236,E2 -17699.236} C_VEL
LIN {X 0,Y 289.737,Z 663.718,A -85,B 0,C 180,E1 -17699.63,E2 -17699.63} C_VEL
LIN {X 0,Y 288.661,Z 674.259,A -85,B 0,C 180,E1 -17700.16,E2 -17700.16} C_VEL
LIN {X 0,Y 287.307,Z 684.335,A -85,B 0,C 180,E1 -17700.811,E2 -17700.811} C_VEL
LIN {X 0,Y 285.589,Z 695.377,A -85,B 0,C 180,E1 -17701.725,E2 -17701.725} C_VEL
LIN {X 0,Y 283.807,Z 705.295,A -85,B 0,C 180,E1 -17702.735,E2 -17702.735} C_VEL
LIN {X 0,Y 281.979,Z 715.049,A -85,B 0,C 180,E1 -17703.947,E2 -17703.947} C_VEL
LIN {X 0,Y 280.013,Z 724.441,A -85,B 0,C 180,E1 -17705.338,E2 -17705.338} C_VEL
LIN {X 0,Y 277.79,Z 733.457,A -85,B 0,C 180,E1 -17706.913,E2 -17706.913} C_VEL
LIN {X 0,Y 276.157,Z 740.433,A -85,B 0,C 180,E1 -17708.346,E2 -17708.346} C_VEL
LIN {X 0,Y 274.293,Z 747.956,A -85,B 0,C 180,E1 -17710.154,E2 -17710.154} C_VEL
LIN {X 0,Y 272.45,Z 755.524,A -85,B 0,C 180,E1 -17712.341,E2 -17712.341} C_VEL
LIN {X 0,Y 271.276,Z 760.976,A -85,B 0,C 180,E1 -17714.216,E2 -17714.216} C_VEL
LIN {X 0,Y 270.037,Z 766.411,A -85,B 0,C 180,E1 -17716.454,E2 -17716.454} C_VEL
LIN {X 0,Y 269.106,Z 770.857,A -85,B 0,C 180,E1 -17718.705,E2 -17718.705} C_VEL
LIN {X 0,Y 268.606,Z 774.407,A -85,B 0,C 180,E1 -17720.968,E2 -17720.968} C_VEL
LIN {X 0,Y 268.34,Z 776.35,A -85,B 0,C 180,E1 -17722.475,E2 -17722.475} C_VEL
LIN {X 0,Y 268.133,Z 779.04,A -85,B 0,C 180,E1 -17725.49,E2 -17725.49} C_VEL
LIN {X 0,Y 268.186,Z 780.336,A -85,B 0,C 180,E1 -17728.498,E2 -17728.498} C_VEL
LIN {X 0,Y 268.202,Z 780.589,A -85,B 0,C 180,E1 -17730,E2 -17730} C_VEL
LIN {X 0,Y 268.154,Z 779.86,A -85,B 0,C 180,E1 -17733.005,E2 -17733.005} C_VEL
LIN {X 0,Y 268.157,Z 778.578,A -85,B 0,C 180,E1 -17735.169,E2 -17735.169} C_VEL
LIN {X 0,Y 268.34,Z 776.35,A -85,B 0,C 180,E1 -17737.525,E2 -17737.525} C_VEL
LIN {X 0,Y 268.734,Z 773.389,A -85,B 0,C 180,E1 -17739.787,E2 -17739.787} C_VEL
LIN {X 0,Y 269.345,Z 769.557,A -85,B 0,C 180,E1 -17742.048,E2 -17742.048} C_VEL
LIN {X 0,Y 270.422,Z 764.795,A -85,B 0,C 180,E1 -17744.294,E2 -17744.294} C_VEL
LIN {X 0,Y 271.915,Z 757.572,A -85,B 0,C 180,E1 -17746.996,E2 -17746.996} C_VEL
LIN {X 0,Y 273.642,Z 750.632,A -85,B 0,C 180,E1 -17749.114,E2 -17749.114} C_VEL
LIN {X 0,Y 275.356,Z 743.556,A -85,B 0,C 180,E1 -17750.936,E2 -17750.936} C_VEL
LIN {X 0,Y 276.894,Z 737.093,A -85,B 0,C 180,E1 -17752.378,E2 -17752.378} C_VEL
LIN {X 0,Y 279.244,Z 727.618,A -85,B 0,C 180,E1 -17754.14,E2 -17754.14} C_VEL
LIN {X 0,Y 281.17,Z 719.374,A -85,B 0,C 180,E1 -17755.441,E2 -17755.441} C_VEL
LIN {X 0,Y 283.016,Z 709.689,A -85,B 0,C 180,E1 -17756.749,E2 -17756.749} C_VEL
LIN {X 0,Y 284.993,Z 698.884,A -85,B 0,C 180,E1 -17757.939,E2 -17757.939} C_VEL
LIN {X 0,Y 286.641,Z 688.627,A -85,B 0,C 180,E1 -17758.862,E2 -17758.862} C_VEL
LIN {X 0,Y 288.278,Z 676.977,A -85,B 0,C 180,E1 -17759.682,E2 -17759.682} C_VEL
LIN {X 0,Y 289.452,Z 666.452,A -85,B 0,C 180,E1 -17760.252,E2 -17760.252} C_VEL
LIN {X 0,Y 290.357,Z 655.339,A -85,B 0,C 180,E1 -17760.69,E2 -17760.69} C_VEL
LIN {X 0,Y 291.614,Z 626.039,A -85,B 0,C 180,E1 -17761.429,E2 -17761.429} C_VEL
LIN {X 0,Y 293.305,Z 574.408,A -85,B 0,C 180,E1 -17762.685,E2 -17762.685} C_VEL
LIN {X 0,Y 289.736,Z 554.854,A -85,B 0,C 180,E1 -17763.704,E2 -17763.704} C_VEL
LIN {X 0,Y 288.634,Z 550.961,A -85,B 0,C 180,E1 -17763.963,E2 -17763.963} C_VEL
LIN {X 0,Y 282.063,Z 536.048,A -85,B 0,C 180,E1 -17765.313,E2 -17765.313} C_VEL
LIN {X 0,Y 274.833,Z 521.382,A -85,B 0,C 180,E1 -17766.847,E2 -17766.847} C_VEL
LIN {X 0,Y 273.01,Z 517.604,A -85,B 0,C 180,E1 -17767.32,E2 -17767.32} C_VEL
LIN {X 0,Y 270.967,Z 509.006,A -85,B 0,C 180,E1 -17771.221,E2 -17771.221} C_VEL
LIN {X 0,Y 270.207,Z 506.023,A -85,B 0,C 180,E1 -17772.722,E2 -17772.722} C_VEL
LIN {X 0,Y 270.19,Z 505.944,A -85,B 0,C 180,E1 -17777.444,E2 -17777.444} C_VEL
LIN {X 0,Y 270.243,Z 505.934,A -85,B 0,C 180,E1 -17781.38,E2 -17781.38} C_VEL
LIN {X 0,Y 270.212,Z 505.946,A -85,B 0,C 180,E1 -17785.095,E2 -17785.095} C_VEL
LIN {X 0,Y 270.197,Z 505.951,A -85,B 0,C 180,E1 -17789.13,E2 -17789.13} C_VEL
LIN {X 0,Y 270.259,Z 505.922,A -85,B 0,C 180,E1 -17792.146,E2 -17792.146} C_VEL
LIN {X 0,Y 270.233,Z 505.948,A -85,B 0,C 180,E1 -17795.537,E2 -17795.537} C_VEL
LIN {X 0,Y 270.296,Z 505.916,A -85,B 0,C 180,E1 -17800.243,E2 -17800.243} C_VEL
LIN {X 0,Y 270.391,Z 505.907,A -85,B 0,C 180,E1 -17804.934,E2 -17804.934} C_VEL
LIN {X 0,Y 270.436,Z 505.92,A -85,B 0,C 180,E1 -17809.518,E2 -17809.518} C_VEL
LIN {X 0,Y 270.602,Z 505.881,A -85,B 0,C 180,E1 -17812.538,E2 -17812.538} C_VEL
LIN {X 0,Y 270.781,Z 505.877,A -85,B 0,C 180,E1 -17818.512,E2 -17818.512} C_VEL
LIN {X 0,Y 270.781,Z 505.844,A -85,B 0,C 180,E1 -17821.487,E2 -17821.487} C_VEL
LIN {X 0,Y 270.592,Z 505.892,A -85,B 0,C 180,E1 -17827.461,E2 -17827.461} C_VEL
LIN {X 0,Y 270.406,Z 505.894,A -85,B 0,C 180,E1 -17830.482,E2 -17830.482} C_VEL
LIN {X 0,Y 270.39,Z 505.921,A -85,B 0,C 180,E1 -17835.065,E2 -17835.065} C_VEL
LIN {X 0,Y 270.295,Z 505.933,A -85,B 0,C 180,E1 -17839.755,E2 -17839.755} C_VEL
LIN {X 0,Y 270.268,Z 505.917,A -85,B 0,C 180,E1 -17844.585,E2 -17844.585} C_VEL
LIN {X 0,Y 270.266,Z 505.944,A -85,B 0,C 180,E1 -17847.908,E2 -17847.908} C_VEL
LIN {X 0,Y 270.179,Z 505.935,A -85,B 0,C 180,E1 -17851.348,E2 -17851.348} C_VEL
LIN {X 0,Y 270.209,Z 505.939,A -85,B 0,C 180,E1 -17854.903,E2 -17854.903} C_VEL
LIN {X 0,Y 270.216,Z 505.952,A -85,B 0,C 180,E1 -17858.717,E2 -17858.717} C_VEL
LIN {X 0,Y 270.225,Z 505.949,A -85,B 0,C 180,E1 -17862.547,E2 -17862.547} C_VEL
LIN {X 0,Y 270.226,Z 505.895,A -85,B 0,C 180,E1 -17866.736,E2 -17866.736} C_VEL
LIN {X 0,Y 270.241,Z 505.928,A -85,B 0,C 180,E1 -17869.447,E2 -17869.447} C_VEL
LIN {X 0,Y 270.267,Z 506.186,A -85,B 0,C 180,E1 -17872.116,E2 -17872.116} C_VEL
LIN {X 0,Y 270.563,Z 507.309,A -85,B 0,C 180,E1 -17872.394,E2 -17872.394} C_VEL
LIN {X 0,Y 272.17,Z 509.956,A -85,B 0,C 180,E1 -17872.756,E2 -17872.756} C_VEL
LIN {X 0,Y 284.308,Z 529.419,A -85,B 0,C 180,E1 -17875.197,E2 -17875.197} C_VEL
LIN {X 0,Y 290.408,Z 537.211,A -85,B 0,C 180,E1 -17876.263,E2 -17876.263} C_VEL
LIN {X 0,Y 299.504,Z 547.375,A -85,B 0,C 180,E1 -17877.771,E2 -17877.771} C_VEL
LIN {X 0,Y 308.314,Z 556.183,A -85,B 0,C 180,E1 -17879.37,E2 -17879.37} C_VEL
LIN {X 0,Y 314.794,Z 562.656,A -85,B 0,C 180,E1 -17880.677,E2 -17880.677} C_VEL
LIN {X 0,Y 321.457,Z 569.176,A -85,B 0,C 180,E1 -17882.171,E2 -17882.171} C_VEL
LIN {X 0,Y 328.819,Z 576.116,A -85,B 0,C 180,E1 -17883.958,E2 -17883.958} C_VEL
LIN {X 0,Y 336.644,Z 583.182,A -85,B 0,C 180,E1 -17885.994,E2 -17885.994} C_VEL
LIN {X 0,Y 340.671,Z 586.641,A -85,B 0,C 180,E1 -17887.107,E2 -17887.107} C_VEL
LIN {X 0,Y 346.134,Z 591.208,A -85,B 0,C 180,E1 -17888.703,E2 -17888.703} C_VEL
LIN {X 0,Y 349.203,Z 593.757,A -85,B 0,C 180,E1 -17889.657,E2 -17889.657} C_VEL
LIN {X 0,Y 354.537,Z 598.241,A -85,B 0,C 180,E1 -17891.431,E2 -17891.431} C_VEL
LIN {X 0,Y 359.166,Z 601.663,A -85,B 0,C 180,E1 -17893.098,E2 -17893.098} C_VEL
LIN {X 0,Y 363.379,Z 605.311,A -85,B 0,C 180,E1 -17894.797,E2 -17894.797} C_VEL
LIN {X 0,Y 367.464,Z 607.965,A -85,B 0,C 180,E1 -17896.605,E2 -17896.605} C_VEL
LIN {X 0,Y 369.721,Z 609.44,A -85,B 0,C 180,E1 -17897.721,E2 -17897.721} C_VEL
LIN {X 0,Y 373.456,Z 612.766,A -85,B 0,C 180,E1 -17899.892,E2 -17899.892} C_VEL
LIN {X 0,Y 376.273,Z 614.698,A -85,B 0,C 180,E1 -17901.857,E2 -17901.857} C_VEL
LIN {X 0,Y 378.817,Z 616.104,A -85,B 0,C 180,E1 -17904.133,E2 -17904.133} C_VEL
LIN {X 0,Y 380.375,Z 616.737,A -85,B 0,C 180,E1 -17906.128,E2 -17906.128} C_VEL
LIN {X 0,Y 381.384,Z 617.221,A -85,B 0,C 180,E1 -17908.416,E2 -17908.416} C_VEL
LIN {X 0,Y 381.625,Z 617.193,A -85,B 0,C 180,E1 -17910,E2 -17910} C_VEL
LIN {X 0,Y 381.384,Z 617.223,A -85,B 0,C 180,E1 -17911.584,E2 -17911.584} C_VEL
LIN {X 0,Y 380.376,Z 616.738,A -85,B 0,C 180,E1 -17913.873,E2 -17913.873} C_VEL
LIN {X 0,Y 378.602,Z 616.007,A -85,B 0,C 180,E1 -17916.083,E2 -17916.083} C_VEL
LIN {X 0,Y 376.272,Z 614.711,A -85,B 0,C 180,E1 -17918.143,E2 -17918.143} C_VEL
LIN {X 0,Y 373.168,Z 612.571,A -85,B 0,C 180,E1 -17920.284,E2 -17920.284} C_VEL
LIN {X 0,Y 369.455,Z 609.137,A -85,B 0,C 180,E1 -17922.426,E2 -17922.426} C_VEL
LIN {X 0,Y 364.781,Z 606.313,A -85,B 0,C 180,E1 -17924.595,E2 -17924.595} C_VEL
LIN {X 0,Y 360.358,Z 602.797,A -85,B 0,C 180,E1 -17926.433,E2 -17926.433} C_VEL
LIN {X 0,Y 356.841,Z 599.795,A -85,B 0,C 180,E1 -17927.766,E2 -17927.766} C_VEL
LIN {X 0,Y 351.663,Z 595.955,A -85,B 0,C 180,E1 -17929.54,E2 -17929.54} C_VEL
LIN {X 0,Y 346.897,Z 591.768,A -85,B 0,C 180,E1 -17931.063,E2 -17931.063} C_VEL
LIN {X 0,Y 341.385,Z 587.317,A -85,B 0,C 180,E1 -17932.688,E2 -17932.688} C_VEL
LIN {X 0,Y 336.928,Z 583.413,A -85,B 0,C 180,E1 -17933.931,E2 -17933.931} C_VEL
LIN {X 0,Y 331.033,Z 578.057,A -85,B 0,C 180,E1 -17935.483,E2 -17935.483} C_VEL
LIN {X 0,Y 324.218,Z 571.846,A -85,B 0,C 180,E1 -17937.169,E2 -17937.169} C_VEL
LIN {X 0,Y 316.711,Z 564.606,A -85,B 0,C 180,E1 -17938.899,E2 -17938.899} C_VEL
LIN {X 0,Y 309.355,Z 557.266,A -85,B 0,C 180,E1 -17940.426,E2 -17940.426} C_VEL
LIN {X 0,Y 301.062,Z 548.943,A -85,B 0,C 180,E1 -17941.962,E2 -17941.962} C_VEL
LIN {X 0,Y 291.611,Z 538.645,A -85,B 0,C 180,E1 -17943.537,E2 -17943.537} C_VEL
LIN {X 0,Y 286.064,Z 531.717,A -85,B 0,C 180,E1 -17944.489,E2 -17944.489} C_VEL
LIN {X 0,Y 280,Z 522.874,A -85,B 0,C 180,E1 -17945.625,E2 -17945.625} C_VEL
LIN {X 0,Y 273.639,Z 512.429,A -85,B 0,C 180,E1 -17946.929,E2 -17946.929} C_VEL
LIN {X 0,Y 272.168,Z 509.984,A -85,B 0,C 180,E1 -17947.243,E2 -17947.243} C_VEL
LIN {X 0,Y 270.565,Z 507.279,A -85,B 0,C 180,E1 -17947.607,E2 -17947.607} C_VEL
LIN {X 0,Y 270.272,Z 506.111,A -85,B 0,C 180,E1 -17947.922,E2 -17947.922} C_VEL
LIN {X 0,Y 270.245,Z 505.915,A -85,B 0,C 180,E1 -17951.048,E2 -17951.048} C_VEL
LIN {X 0,Y 270.225,Z 505.921,A -85,B 0,C 180,E1 -17955.396,E2 -17955.396} C_VEL
LIN {X 0,Y 270.24,Z 505.932,A -85,B 0,C 180,E1 -17959.447,E2 -17959.447} C_VEL
LIN {X 0,Y 270.25,Z 505.928,A -85,B 0,C 180,E1 -17963.722,E2 -17963.722} C_VEL
LIN {X 0,Y 270.199,Z 505.953,A -85,B 0,C 180,E1 -17966.893,E2 -17966.893} C_VEL
LIN {X 0,Y 270.223,Z 505.929,A -85,B 0,C 180,E1 -17970.387,E2 -17970.387} C_VEL
LIN {X 0,Y 270.257,Z 505.935,A -85,B 0,C 180,E1 -17973.764,E2 -17973.764} C_VEL
LIN {X 0,Y 270.225,Z 505.93,A -85,B 0,C 180,E1 -17977.039,E2 -17977.039} C_VEL
LIN {X 0,Y 270.295,Z 505.933,A -85,B 0,C 180,E1 -17980.245,E2 -17980.245} C_VEL
LIN {X 0,Y 270.39,Z 505.921,A -85,B 0,C 180,E1 -17984.935,E2 -17984.935} C_VEL
LIN {X 0,Y 270.406,Z 505.894,A -85,B 0,C 180,E1 -17989.518,E2 -17989.518} C_VEL
LIN {X 0,Y 270.593,Z 505.892,A -85,B 0,C 180,E1 -17992.539,E2 -17992.539} C_VEL
LIN {X 0,Y 270.781,Z 505.844,A -85,B 0,C 180,E1 -17998.513,E2 -17998.513} C_VEL
LIN {X 0,Y 270.781,Z 505.877,A -85,B 0,C 180,E1 -18001.488,E2 -18001.488} C_VEL
LIN {X 0,Y 270.602,Z 505.881,A -85,B 0,C 180,E1 -18007.462,E2 -18007.462} C_VEL
LIN {X 0,Y 270.436,Z 505.92,A -85,B 0,C 180,E1 -18010.482,E2 -18010.482} C_VEL
LIN {X 0,Y 270.391,Z 505.907,A -85,B 0,C 180,E1 -18015.066,E2 -18015.066} C_VEL
LIN {X 0,Y 270.296,Z 505.916,A -85,B 0,C 180,E1 -18019.757,E2 -18019.757} C_VEL
LIN {X 0,Y 270.234,Z 505.947,A -85,B 0,C 180,E1 -18024.59,E2 -18024.59} C_VEL
LIN {X 0,Y 270.266,Z 505.921,A -85,B 0,C 180,E1 -18027.91,E2 -18027.91} C_VEL
LIN {X 0,Y 270.181,Z 505.949,A -85,B 0,C 180,E1 -18031.349,E2 -18031.349} C_VEL
LIN {X 0,Y 270.177,Z 505.935,A -85,B 0,C 180,E1 -18032.761,E2 -18032.761} C_VEL
LIN {X 0,Y 269.563,Z 506.016,A -85,B 0,C 180,E1 -18034.006,E2 -18034.006} C_VEL
LIN {X 0,Y 266.73,Z 506.386,A -85,B 0,C 180,E1 -18036.035,E2 -18036.035} C_VEL
LIN {X 0,Y 264.289,Z 506.683,A -85,B 0,C 180,E1 -18037.685,E2 -18037.685} C_VEL
LIN {X 0,Y 263.236,Z 506.812,A -85,B 0,C 180,E1 -18038.964,E2 -18038.964} C_VEL
LIN {X 0,Y 263.149,Z 506.827,A -85,B 0,C 180,E1 -18039.398,E2 -18039.398} C_VEL
LIN {X 0,Y 263.141,Z 506.822,A -85,B 0,C 180,E1 -18041.891,E2 -18041.891} C_VEL
LIN {X 0,Y 263.133,Z 506.953,A -85,B 0,C 180,E1 -18046.426,E2 -18046.426} C_VEL
LIN {X 0,Y 265.065,Z 514.599,A -85,B 0,C 180,E1 -18050.257,E2 -18050.257} C_VEL
LIN {X 0,Y 265.759,Z 517.479,A -85,B 0,C 180,E1 -18051.5,E2 -18051.5} C_VEL
LIN {X 0,Y 272.956,Z 531.5,A -85,B 0,C 180,E1 -18053.185,E2 -18053.185} C_VEL
LIN {X 0,Y 280.774,Z 548.341,A -85,B 0,C 180,E1 -18054.878,E2 -18054.878} C_VEL
LIN {X 0,Y 283.698,Z 555.844,A -85,B 0,C 180,E1 -18055.515,E2 -18055.515} C_VEL
LIN {X 0,Y 287.321,Z 575.615,A -85,B 0,C 180,E1 -18056.587,E2 -18056.587} C_VEL
LIN {X 0,Y 284.525,Z 651.749,A -85,B 0,C 180,E1 -18058.476,E2 -18058.476} C_VEL
LIN {X 0,Y 283.639,Z 663.52,A -85,B 0,C 180,E1 -18058.905,E2 -18058.905} C_VEL
LIN {X 0,Y 282.525,Z 674.061,A -85,B 0,C 180,E1 -18059.444,E2 -18059.444} C_VEL
LIN {X 0,Y 281.105,Z 684.137,A -85,B 0,C 180,E1 -18060.102,E2 -18060.102} C_VEL
LIN {X 0,Y 279.339,Z 695.179,A -85,B 0,C 180,E1 -18061.033,E2 -18061.033} C_VEL
LIN {X 0,Y 277.497,Z 705.096,A -85,B 0,C 180,E1 -18062.061,E2 -18062.061} C_VEL
LIN {X 0,Y 275.576,Z 714.85,A -85,B 0,C 180,E1 -18063.294,E2 -18063.294} C_VEL
LIN {X 0,Y 273.563,Z 724.243,A -85,B 0,C 180,E1 -18064.717,E2 -18064.717} C_VEL
LIN {X 0,Y 271.253,Z 733.258,A -85,B 0,C 180,E1 -18066.323,E2 -18066.323} C_VEL
LIN {X 0,Y 269.521,Z 740.233,A -85,B 0,C 180,E1 -18067.784,E2 -18067.784} C_VEL
LIN {X 0,Y 267.585,Z 747.756,A -85,B 0,C 180,E1 -18069.635,E2 -18069.635} C_VEL
LIN {X 0,Y 265.941,Z 754.232,A -85,B 0,C 180,E1 -18071.511,E2 -18071.511} C_VEL
LIN {X 0,Y 264.396,Z 760.777,A -85,B 0,C 180,E1 -18073.794,E2 -18073.794} C_VEL
LIN {X 0,Y 263.095,Z 766.211,A -85,B 0,C 180,E1 -18076.089,E2 -18076.089} C_VEL
LIN {X 0,Y 262.097,Z 770.657,A -85,B 0,C 180,E1 -18078.398,E2 -18078.398} C_VEL
LIN {X 0,Y 261.546,Z 774.208,A -85,B 0,C 180,E1 -18080.722,E2 -18080.722} C_VEL
LIN {X 0,Y 261.285,Z 776.151,A -85,B 0,C 180,E1 -18082.271,E2 -18082.271} C_VEL
LIN {X 0,Y 261.048,Z 778.842,A -85,B 0,C 180,E1 -18085.367,E2 -18085.367} C_VEL
LIN {X 0,Y 261.113,Z 780.139,A -85,B 0,C 180,E1 -18088.458,E2 -18088.458} C_VEL
LIN {X 0,Y 261.127,Z 780.392,A -85,B 0,C 180,E1 -18090,E2 -18090} C_VEL
LIN {X 0,Y 261.049,Z 779.662,A -85,B 0,C 180,E1 -18093.086,E2 -18093.086} C_VEL
LIN {X 0,Y 261.051,Z 778.596,A -85,B 0,C 180,E1 -18095.05,E2 -18095.05} C_VEL
LIN {X 0,Y 261.285,Z 776.151,A -85,B 0,C 180,E1 -18097.729,E2 -18097.729} C_VEL
LIN {X 0,Y 261.885,Z 771.926,A -85,B 0,C 180,E1 -18100.827,E2 -18100.827} C_VEL
LIN {X 0,Y 262.715,Z 767.79,A -85,B 0,C 180,E1 -18103.143,E2 -18103.143} C_VEL
LIN {X 0,Y 263.889,Z 762.689,A -85,B 0,C 180,E1 -18105.445,E2 -18105.445} C_VEL
LIN {X 0,Y 265.307,Z 756.509,A -85,B 0,C 180,E1 -18107.735,E2 -18107.735} C_VEL
LIN {X 0,Y 266.888,Z 750.432,A -85,B 0,C 180,E1 -18109.618,E2 -18109.618} C_VEL
LIN {X 0,Y 268.688,Z 743.356,A -85,B 0,C 180,E1 -18111.481,E2 -18111.481} C_VEL
LIN {X 0,Y 270.305,Z 736.894,A -85,B 0,C 180,E1 -18112.954,E2 -18112.954} C_VEL
LIN {X 0,Y 272.749,Z 727.419,A -85,B 0,C 180,E1 -18114.753,E2 -18114.753} C_VEL
LIN {X 0,Y 275.042,Z 717.752,A -85,B 0,C 180,E1 -18116.283,E2 -18116.283} C_VEL
LIN {X 0,Y 276.682,Z 709.491,A -85,B 0,C 180,E1 -18117.412,E2 -18117.412} C_VEL
LIN {X 0,Y 278.743,Z 698.687,A -85,B 0,C 180,E1 -18118.623,E2 -18118.623} C_VEL
LIN {X 0,Y 280.449,Z 688.43,A -85,B 0,C 180,E1 -18119.561,E2 -18119.561} C_VEL
LIN {X 0,Y 282.135,Z 676.779,A -85,B 0,C 180,E1 -18120.396,E2 -18120.396} C_VEL
LIN {X 0,Y 283.432,Z 665.343,A -85,B 0,C 180,E1 -18121.016,E2 -18121.016} C_VEL
LIN {X 0,Y 284.335,Z 654.028,A -85,B 0,C 180,E1 -18121.455,E2 -18121.455} C_VEL
LIN {X 0,Y 285.898,Z 617.245,A -85,B 0,C 180,E1 -18122.382,E2 -18122.382} C_VEL
LIN {X 0,Y 287.284,Z 575.534,A -85,B 0,C 180,E1 -18123.421,E2 -18123.421} C_VEL
LIN {X 0,Y 284.002,Z 557.157,A -85,B 0,C 180,E1 -18124.404,E2 -18124.404} C_VEL
LIN {X 0,Y 282.832,Z 553.368,A -85,B 0,C 180,E1 -18124.68,E2 -18124.68} C_VEL
LIN {X 0,Y 276.688,Z 539.35,A -85,B 0,C 180,E1 -18125.996,E2 -18125.996} C_VEL
LIN {X 0,Y 269.927,Z 525.54,A -85,B 0,C 180,E1 -18127.489,E2 -18127.489} C_VEL
LIN {X 0,Y 265.752,Z 517.495,A -85,B 0,C 180,E1 -18128.498,E2 -18128.498} C_VEL
LIN {X 0,Y 264.564,Z 512.437,A -85,B 0,C 180,E1 -18130.792,E2 -18130.792} C_VEL
LIN {X 0,Y 263.129,Z 506.828,A -85,B 0,C 180,E1 -18133.71,E2 -18133.71} C_VEL
LIN {X 0,Y 263.141,Z 506.82,A -85,B 0,C 180,E1 -18138.109,E2 -18138.109} C_VEL
LIN {X 0,Y 263.186,Z 506.811,A -85,B 0,C 180,E1 -18142.107,E2 -18142.107} C_VEL
LIN {X 0,Y 263.182,Z 506.811,A -85,B 0,C 180,E1 -18145.889,E2 -18145.889} C_VEL
LIN {X 0,Y 263.138,Z 506.833,A -85,B 0,C 180,E1 -18149.504,E2 -18149.504} C_VEL
LIN {X 0,Y 263.185,Z 506.8,A -85,B 0,C 180,E1 -18153.001,E2 -18153.001} C_VEL
LIN {X 0,Y 263.151,Z 506.83,A -85,B 0,C 180,E1 -18156.383,E2 -18156.383} C_VEL
LIN {X 0,Y 263.258,Z 506.788,A -85,B 0,C 180,E1 -18159.692,E2 -18159.692} C_VEL
LIN {X 0,Y 263.34,Z 506.792,A -85,B 0,C 180,E1 -18164.521,E2 -18164.521} C_VEL
LIN {X 0,Y 263.368,Z 506.798,A -85,B 0,C 180,E1 -18169.233,E2 -18169.233} C_VEL
LIN {X 0,Y 263.564,Z 506.76,A -85,B 0,C 180,E1 -18172.337,E2 -18172.337} C_VEL
LIN {X 0,Y 263.745,Z 506.753,A -85,B 0,C 180,E1 -18178.472,E2 -18178.472} C_VEL
LIN {X 0,Y 263.745,Z 506.719,A -85,B 0,C 180,E1 -18181.526,E2 -18181.526} C_VEL
LIN {X 0,Y 263.552,Z 506.767,A -85,B 0,C 180,E1 -18187.661,E2 -18187.661} C_VEL
LIN {X 0,Y 263.349,Z 506.774,A -85,B 0,C 180,E1 -18190.766,E2 -18190.766} C_VEL
LIN {X 0,Y 263.338,Z 506.793,A -85,B 0,C 180,E1 -18195.478,E2 -18195.478} C_VEL
LIN {X 0,Y 263.257,Z 506.817,A -85,B 0,C 180,E1 -18200.306,E2 -18200.306} C_VEL
LIN {X 0,Y 263.202,Z 506.801,A -85,B 0,C 180,E1 -18205.291,E2 -18205.291} C_VEL
LIN {X 0,Y 263.174,Z 506.819,A -85,B 0,C 180,E1 -18208.729,E2 -18208.729} C_VEL
LIN {X 0,Y 263.128,Z 506.824,A -85,B 0,C 180,E1 -18212.288,E2 -18212.288} C_VEL
LIN {X 0,Y 263.182,Z 506.808,A -85,B 0,C 180,E1 -18215.978,E2 -18215.978} C_VEL
LIN {X 0,Y 263.154,Z 506.819,A -85,B 0,C 180,E1 -18219.862,E2 -18219.862} C_VEL
LIN {X 0,Y 263.185,Z 506.813,A -85,B 0,C 180,E1 -18223.97,E2 -18223.97} C_VEL
LIN {X 0,Y 263.166,Z 506.782,A -85,B 0,C 180,E1 -18228.116,E2 -18228.116} C_VEL
LIN {X 0,Y 263.217,Z 506.979,A -85,B 0,C 180,E1 -18230.884,E2 -18230.884} C_VEL
LIN {X 0,Y 263.487,Z 508.036,A -85,B 0,C 180,E1 -18231.209,E2 -18231.209} C_VEL
LIN {X 0,Y 264.968,Z 510.695,A -85,B 0,C 180,E1 -18231.579,E2 -18231.579} C_VEL
LIN {X 0,Y 266.335,Z 512.747,A -85,B 0,C 180,E1 -18231.883,E2 -18231.883} C_VEL
LIN {X 0,Y 273.462,Z 524.39,A -85,B 0,C 180,E1 -18233.428,E2 -18233.428} C_VEL
LIN {X 0,Y 280.958,Z 535.833,A -85,B 0,C 180,E1 -18234.914,E2 -18234.914} C_VEL
LIN {X 0,Y 286.143,Z 542.479,A -85,B 0,C 180,E1 -18235.843,E2 -18235.843} C_VEL
LIN {X 0,Y 296.297,Z 553.666,A -85,B 0,C 180,E1 -18237.512,E2 -18237.512} C_VEL
LIN {X 0,Y 304.718,Z 561.923,A -85,B 0,C 180,E1 -18238.974,E2 -18238.974} C_VEL
LIN {X 0,Y 311.463,Z 568.54,A -85,B 0,C 180,E1 -18240.281,E2 -18240.281} C_VEL
LIN {X 0,Y 318.31,Z 575.1,A -85,B 0,C 180,E1 -18241.743,E2 -18241.743} C_VEL
LIN {X 0,Y 325.9,Z 582.153,A -85,B 0,C 180,E1 -18243.533,E2 -18243.533} C_VEL
LIN {X 0,Y 334.066,Z 589.413,A -85,B 0,C 180,E1 -18245.609,E2 -18245.609} C_VEL
LIN {X 0,Y 338.301,Z 593.01,A -85,B 0,C 180,E1 -18246.752,E2 -18246.752} C_VEL
LIN {X 0,Y 343.9,Z 597.635,A -85,B 0,C 180,E1 -18248.356,E2 -18248.356} C_VEL
LIN {X 0,Y 348.428,Z 601.412,A -85,B 0,C 180,E1 -18249.746,E2 -18249.746} C_VEL
LIN {X 0,Y 354.133,Z 605.864,A -85,B 0,C 180,E1 -18251.635,E2 -18251.635} C_VEL
LIN {X 0,Y 357.718,Z 608.605,A -85,B 0,C 180,E1 -18252.92,E2 -18252.92} C_VEL
LIN {X 0,Y 362.315,Z 612.417,A -85,B 0,C 180,E1 -18254.752,E2 -18254.752} C_VEL
LIN {X 0,Y 366.45,Z 614.998,A -85,B 0,C 180,E1 -18256.567,E2 -18256.567} C_VEL
LIN {X 0,Y 368.732,Z 616.589,A -85,B 0,C 180,E1 -18257.687,E2 -18257.687} C_VEL
LIN {X 0,Y 372.217,Z 619.642,A -85,B 0,C 180,E1 -18259.685,E2 -18259.685} C_VEL
LIN {X 0,Y 375.171,Z 621.651,A -85,B 0,C 180,E1 -18261.704,E2 -18261.704} C_VEL
LIN {X 0,Y 377.707,Z 623.039,A -85,B 0,C 180,E1 -18263.902,E2 -18263.902} C_VEL
LIN {X 0,Y 379.249,Z 623.721,A -85,B 0,C 180,E1 -18265.749,E2 -18265.749} C_VEL
LIN {X 0,Y 380.378,Z 624.136,A -85,B 0,C 180,E1 -18267.882,E2 -18267.882} C_VEL
LIN {X 0,Y 380.648,Z 624.347,A -85,B 0,C 180,E1 -18268.942,E2 -18268.942} C_VEL
LIN {X 0,Y 380.761,Z 624.231,A -85,B 0,C 180,E1 -18270,E2 -18270} C_VEL
LIN {X 0,Y 380.515,Z 624.27,A -85,B 0,C 180,E1 -18271.588,E2 -18271.588} C_VEL
LIN {X 0,Y 379.917,Z 623.895,A -85,B 0,C 180,E1 -18273.181,E2 -18273.181} C_VEL
LIN {X 0,Y 378.41,Z 623.392,A -85,B 0,C 180,E1 -18275.328,E2 -18275.328} C_VEL
LIN {X 0,Y 376.145,Z 622.252,A -85,B 0,C 180,E1 -18277.515,E2 -18277.515} C_VEL
LIN {X 0,Y 373.215,Z 620.361,A -85,B 0,C 180,E1 -18279.668,E2 -18279.668} C_VEL
LIN {X 0,Y 370.283,Z 617.959,A -85,B 0,C 180,E1 -18281.461,E2 -18281.461} C_VEL
LIN {X 0,Y 367.039,Z 615.306,A -85,B 0,C 180,E1 -18283.158,E2 -18283.158} C_VEL
LIN {X 0,Y 362.644,Z 612.655,A -85,B 0,C 180,E1 -18285.109,E2 -18285.109} C_VEL
LIN {X 0,Y 357.712,Z 608.636,A -85,B 0,C 180,E1 -18287.08,E2 -18287.08} C_VEL
LIN {X 0,Y 354.701,Z 606.233,A -85,B 0,C 180,E1 -18288.171,E2 -18288.171} C_VEL
LIN {X 0,Y 349.408,Z 602.263,A -85,B 0,C 180,E1 -18289.939,E2 -18289.939} C_VEL
LIN {X 0,Y 344.174,Z 597.831,A -85,B 0,C 180,E1 -18291.565,E2 -18291.565} C_VEL
LIN {X 0,Y 338.686,Z 593.338,A -85,B 0,C 180,E1 -18293.141,E2 -18293.141} C_VEL
LIN {X 0,Y 333.475,Z 588.915,A -85,B 0,C 180,E1 -18294.546,E2 -18294.546} C_VEL
LIN {X 0,Y 325.045,Z 581.402,A -85,B 0,C 180,E1 -18296.676,E2 -18296.676} C_VEL
LIN {X 0,Y 316.869,Z 573.805,A -85,B 0,C 180,E1 -18298.576,E2 -18298.576} C_VEL
LIN {X 0,Y 308.23,Z 565.518,A -85,B 0,C 180,E1 -18300.353,E2 -18300.353} C_VEL
LIN {X 0,Y 299.668,Z 556.937,A -85,B 0,C 180,E1 -18301.921,E2 -18301.921} C_VEL
LIN {X 0,Y 293.249,Z 550.354,A -85,B 0,C 180,E1 -18302.987,E2 -18302.987} C_VEL
LIN {X 0,Y 284.272,Z 540.346,A -85,B 0,C 180,E1 -18304.479,E2 -18304.479} C_VEL
LIN {X 0,Y 276.782,Z 529.786,A -85,B 0,C 180,E1 -18305.89,E2 -18305.89} C_VEL
LIN {X 0,Y 267.352,Z 514.366,A -85,B 0,C 180,E1 -18307.891,E2 -18307.891} C_VEL
LIN {X 0,Y 265.282,Z 511.008,A -85,B 0,C 180,E1 -18308.356,E2 -18308.356} C_VEL
LIN {X 0,Y 263.606,Z 508.425,A -85,B 0,C 180,E1 -18308.746,E2 -18308.746} C_VEL
LIN {X 0,Y 263.244,Z 507.154,A -85,B 0,C 180,E1 -18309.017,E2 -18309.017} C_VEL
LIN {X 0,Y 263.187,Z 506.825,A -85,B 0,C 180,E1 -18309.857,E2 -18309.857} C_VEL
LIN {X 0,Y 263.185,Z 506.775,A -85,B 0,C 180,E1 -18313.97,E2 -18313.97} C_VEL
LIN {X 0,Y 263.165,Z 506.818,A -85,B 0,C 180,E1 -18318.116,E2 -18318.116} C_VEL
LIN {X 0,Y 263.182,Z 506.824,A -85,B 0,C 180,E1 -18322.108,E2 -18322.108} C_VEL
LIN {X 0,Y 263.178,Z 506.824,A -85,B 0,C 180,E1 -18325.89,E2 -18325.89} C_VEL
LIN {X 0,Y 263.144,Z 506.807,A -85,B 0,C 180,E1 -18329.507,E2 -18329.507} C_VEL
LIN {X 0,Y 263.187,Z 506.825,A -85,B 0,C 180,E1 -18333.003,E2 -18333.003} C_VEL
LIN {X 0,Y 263.177,Z 506.801,A -85,B 0,C 180,E1 -18336.387,E2 -18336.387} C_VEL
LIN {X 0,Y 263.257,Z 506.817,A -85,B 0,C 180,E1 -18339.694,E2 -18339.694} C_VEL
LIN {X 0,Y 263.338,Z 506.793,A -85,B 0,C 180,E1 -18344.522,E2 -18344.522} C_VEL
LIN {X 0,Y 263.349,Z 506.774,A -85,B 0,C 180,E1 -18349.234,E2 -18349.234} C_VEL
LIN {X 0,Y 263.553,Z 506.767,A -85,B 0,C 180,E1 -18352.339,E2 -18352.339} C_VEL
LIN {X 0,Y 263.745,Z 506.719,A -85,B 0,C 180,E1 -18358.474,E2 -18358.474} C_VEL
LIN {X 0,Y 263.745,Z 506.753,A -85,B 0,C 180,E1 -18361.528,E2 -18361.528} C_VEL
LIN {X 0,Y 263.564,Z 506.76,A -85,B 0,C 180,E1 -18367.663,E2 -18367.663} C_VEL
LIN {X 0,Y 263.368,Z 506.798,A -85,B 0,C 180,E1 -18370.767,E2 -18370.767} C_VEL
LIN {X 0,Y 263.34,Z 506.792,A -85,B 0,C 180,E1 -18375.479,E2 -18375.479} C_VEL
LIN {X 0,Y 263.258,Z 506.788,A -85,B 0,C 180,E1 -18380.308,E2 -18380.308} C_VEL
LIN {X 0,Y 263.188,Z 506.818,A -85,B 0,C 180,E1 -18385.294,E2 -18385.294} C_VEL
LIN {X 0,Y 263.162,Z 506.815,A -85,B 0,C 180,E1 -18388.732,E2 -18388.732} C_VEL
LIN {X 0,Y 263.118,Z 506.814,A -85,B 0,C 180,E1 -18392.759,E2 -18392.759} C_VEL
LIN {X 0,Y 263.201,Z 506.816,A -85,B 0,C 180,E1 -18396.77,E2 -18396.77} C_VEL
LIN {X 0,Y 263.149,Z 506.827,A -85,B 0,C 180,E1 -18399.398,E2 -18399.398} C_VEL
LIN {X 0,Y 262.467,Z 506.921,A -85,B 0,C 180,E1 -18400.248,E2 -18400.248} C_VEL
LIN {X 0,Y 259.615,Z 507.28,A -85,B 0,C 180,E1 -18401.581,E2 -18401.581} C_VEL
LIN {X 0,Y 256.738,Z 507.631,A -85,B 0,C 180,E1 -18402.942,E2 -18402.942} C_VEL
LIN {X 0,Y 256.051,Z 507.709,A -85,B 0,C 180,E1 -18403.824,E2 -18403.824} C_VEL
LIN {X 0,Y 256.086,Z 507.922,A -85,B 0,C 180,E1 -18405.525,E2 -18405.525} C_VEL
LIN {X 0,Y 258.126,Z 515.866,A -85,B 0,C 180,E1 -18409.673,E2 -18409.673} C_VEL
LIN {X 0,Y 258.548,Z 517.452,A -85,B 0,C 180,E1 -18410.249,E2 -18410.249} C_VEL
LIN {X 0,Y 266.222,Z 531.996,A -85,B 0,C 180,E1 -18412.117,E2 -18412.117} C_VEL
LIN {X 0,Y 271.917,Z 543.815,A -85,B 0,C 180,E1 -18413.419,E2 -18413.419} C_VEL
LIN {X 0,Y 278.003,Z 557.982,A -85,B 0,C 180,E1 -18414.777,E2 -18414.777} C_VEL
LIN {X 0,Y 281.392,Z 576.711,A -85,B 0,C 180,E1 -18415.826,E2 -18415.826} C_VEL
LIN {X 0,Y 278.478,Z 651.761,A -85,B 0,C 180,E1 -18417.718,E2 -18417.718} C_VEL
LIN {X 0,Y 277.581,Z 663.322,A -85,B 0,C 180,E1 -18418.148,E2 -18418.148} C_VEL
LIN {X 0,Y 276.428,Z 673.863,A -85,B 0,C 180,E1 -18418.695,E2 -18418.695} C_VEL
LIN {X 0,Y 274.974,Z 683.939,A -85,B 0,C 180,E1 -18419.365,E2 -18419.365} C_VEL
LIN {X 0,Y 273.149,Z 694.981,A -85,B 0,C 180,E1 -18420.312,E2 -18420.312} C_VEL
LIN {X 0,Y 271.228,Z 704.898,A -85,B 0,C 180,E1 -18421.357,E2 -18421.357} C_VEL
LIN {X 0,Y 269.015,Z 715.576,A -85,B 0,C 180,E1 -18422.746,E2 -18422.746} C_VEL
LIN {X 0,Y 267.143,Z 724.044,A -85,B 0,C 180,E1 -18424.064,E2 -18424.064} C_VEL
LIN {X 0,Y 264.752,Z 733.06,A -85,B 0,C 180,E1 -18425.704,E2 -18425.704} C_VEL
LIN {X 0,Y 262.897,Z 740.033,A -85,B 0,C 180,E1 -18427.194,E2 -18427.194} C_VEL
LIN {X 0,Y 260.881,Z 747.557,A -85,B 0,C 180,E1 -18429.088,E2 -18429.088} C_VEL
LIN {X 0,Y 259.154,Z 754.032,A -85,B 0,C 180,E1 -18431.009,E2 -18431.009} C_VEL
LIN {X 0,Y 257.521,Z 760.577,A -85,B 0,C 180,E1 -18433.349,E2 -18433.349} C_VEL
LIN {X 0,Y 256.17,Z 766.012,A -85,B 0,C 180,E1 -18435.705,E2 -18435.705} C_VEL
LIN {X 0,Y 255.105,Z 770.458,A -85,B 0,C 180,E1 -18438.076,E2 -18438.076} C_VEL
LIN {X 0,Y 254.504,Z 774.009,A -85,B 0,C 180,E1 -18440.463,E2 -18440.463} C_VEL
LIN {X 0,Y 254.224,Z 775.952,A -85,B 0,C 180,E1 -18442.055,E2 -18442.055} C_VEL
LIN {X 0,Y 253.975,Z 778.644,A -85,B 0,C 180,E1 -18445.238,E2 -18445.238} C_VEL
LIN {X 0,Y 254.018,Z 779.941,A -85,B 0,C 180,E1 -18448.415,E2 -18448.415} C_VEL
LIN {X 0,Y 254.055,Z 780.194,A -85,B 0,C 180,E1 -18450,E2 -18450} C_VEL
LIN {X 0,Y 253.948,Z 779.464,A -85,B 0,C 180,E1 -18453.173,E2 -18453.173} C_VEL
LIN {X 0,Y 253.954,Z 778.55,A -85,B 0,C 180,E1 -18454.941,E2 -18454.941} C_VEL
LIN {X 0,Y 254.224,Z 775.952,A -85,B 0,C 180,E1 -18457.945,E2 -18457.945} C_VEL
LIN {X 0,Y 254.663,Z 772.991,A -85,B 0,C 180,E1 -18460.334,E2 -18460.334} C_VEL
LIN {X 0,Y 255.379,Z 769.159,A -85,B 0,C 180,E1 -18462.718,E2 -18462.718} C_VEL
LIN {X 0,Y 256.577,Z 764.396,A -85,B 0,C 180,E1 -18465.083,E2 -18465.083} C_VEL
LIN {X 0,Y 258.028,Z 758.187,A -85,B 0,C 180,E1 -18467.576,E2 -18467.576} C_VEL
LIN {X 0,Y 259.817,Z 751.57,A -85,B 0,C 180,E1 -18469.762,E2 -18469.762} C_VEL
LIN {X 0,Y 261.665,Z 744.72,A -85,B 0,C 180,E1 -18471.672,E2 -18471.672} C_VEL
LIN {X 0,Y 263.751,Z 736.695,A -85,B 0,C 180,E1 -18473.559,E2 -18473.559} C_VEL
LIN {X 0,Y 266.303,Z 727.221,A -85,B 0,C 180,E1 -18475.394,E2 -18475.394} C_VEL
LIN {X 0,Y 268.573,Z 717.992,A -85,B 0,C 180,E1 -18476.893,E2 -18476.893} C_VEL
LIN {X 0,Y 270.376,Z 709.292,A -85,B 0,C 180,E1 -18478.107,E2 -18478.107} C_VEL
LIN {X 0,Y 272.516,Z 698.488,A -85,B 0,C 180,E1 -18479.34,E2 -18479.34} C_VEL
LIN {X 0,Y 274.282,Z 688.231,A -85,B 0,C 180,E1 -18480.295,E2 -18480.295} C_VEL
LIN {X 0,Y 276.048,Z 676.581,A -85,B 0,C 180,E1 -18481.14,E2 -18481.14} C_VEL
LIN {X 0,Y 277.291,Z 666.057,A -85,B 0,C 180,E1 -18481.729,E2 -18481.729} C_VEL
LIN {X 0,Y 278.216,Z 655.16,A -85,B 0,C 180,E1 -18482.177,E2 -18482.177} C_VEL
LIN {X 0,Y 279.479,Z 629.306,A -85,B 0,C 180,E1 -18482.852,E2 -18482.852} C_VEL
LIN {X 0,Y 281.383,Z 576.834,A -85,B 0,C 180,E1 -18484.172,E2 -18484.172} C_VEL
LIN {X 0,Y 278.143,Z 558.733,A -85,B 0,C 180,E1 -18485.18,E2 -18485.18} C_VEL
LIN {X 0,Y 273.064,Z 546.273,A -85,B 0,C 180,E1 -18486.325,E2 -18486.325} C_VEL
LIN {X 0,Y 265.247,Z 530.05,A -85,B 0,C 180,E1 -18488.111,E2 -18488.111} C_VEL
LIN {X 0,Y 259.994,Z 520.431,A -85,B 0,C 180,E1 -18489.354,E2 -18489.354} C_VEL
LIN {X 0,Y 258.398,Z 516.972,A -85,B 0,C 180,E1 -18489.861,E2 -18489.861} C_VEL
LIN {X 0,Y 256.564,Z 509.658,A -85,B 0,C 180,E1 -18493.534,E2 -18493.534} C_VEL
LIN {X 0,Y 256.04,Z 507.71,A -85,B 0,C 180,E1 -18494.69,E2 -18494.69} C_VEL
LIN {X 0,Y 256.081,Z 507.703,A -85,B 0,C 180,E1 -18498.801,E2 -18498.801} C_VEL
LIN {X 0,Y 256.152,Z 507.691,A -85,B 0,C 180,E1 -18502.87,E2 -18502.87} C_VEL
LIN {X 0,Y 256.083,Z 507.689,A -85,B 0,C 180,E1 -18506.709,E2 -18506.709} C_VEL
LIN {X 0,Y 256.123,Z 507.689,A -85,B 0,C 180,E1 -18511.409,E2 -18511.409} C_VEL
LIN {X 0,Y 256.139,Z 507.705,A -85,B 0,C 180,E1 -18515.696,E2 -18515.696} C_VEL
LIN {X 0,Y 256.158,Z 507.671,A -85,B 0,C 180,E1 -18519.103,E2 -18519.103} C_VEL
LIN {X 0,Y 256.29,Z 507.678,A -85,B 0,C 180,E1 -18524.084,E2 -18524.084} C_VEL
LIN {X 0,Y 256.304,Z 507.676,A -85,B 0,C 180,E1 -18528.933,E2 -18528.933} C_VEL
LIN {X 0,Y 256.532,Z 507.639,A -85,B 0,C 180,E1 -18532.126,E2 -18532.126} C_VEL
LIN {X 0,Y 256.708,Z 507.63,A -85,B 0,C 180,E1 -18538.43,E2 -18538.43} C_VEL
LIN {X 0,Y 256.708,Z 507.595,A -85,B 0,C 180,E1 -18541.568,E2 -18541.568} C_VEL
LIN {X 0,Y 256.465,Z 507.654,A -85,B 0,C 180,E1 -18546.727,E2 -18546.727} C_VEL
LIN {X 0,Y 256.421,Z 507.633,A -85,B 0,C 180,E1 -18549.464,E2 -18549.464} C_VEL
LIN {X 0,Y 256.245,Z 507.689,A -85,B 0,C 180,E1 -18554.29,E2 -18554.29} C_VEL
LIN {X 0,Y 256.197,Z 507.665,A -85,B 0,C 180,E1 -18557.562,E2 -18557.562} C_VEL
LIN {X 0,Y 256.151,Z 507.703,A -85,B 0,C 180,E1 -18561.119,E2 -18561.119} C_VEL
LIN {X 0,Y 256.182,Z 507.673,A -85,B 0,C 180,E1 -18565.138,E2 -18565.138} C_VEL
LIN {X 0,Y 256.108,Z 507.687,A -85,B 0,C 180,E1 -18569.599,E2 -18569.599} C_VEL
LIN {X 0,Y 256.079,Z 507.712,A -85,B 0,C 180,E1 -18573.29,E2 -18573.29} C_VEL
LIN {X 0,Y 256.134,Z 507.693,A -85,B 0,C 180,E1 -18577.278,E2 -18577.278} C_VEL
LIN {X 0,Y 256.099,Z 507.693,A -85,B 0,C 180,E1 -18581.193,E2 -18581.193} C_VEL
LIN {X 0,Y 256.111,Z 507.679,A -85,B 0,C 180,E1 -18584.483,E2 -18584.483} C_VEL
LIN {X 0,Y 256.127,Z 507.654,A -85,B 0,C 180,E1 -18587.804,E2 -18587.804} C_VEL
LIN {X 0,Y 256.167,Z 507.943,A -85,B 0,C 180,E1 -18589.662,E2 -18589.662} C_VEL
LIN {X 0,Y 256.45,Z 509.086,A -85,B 0,C 180,E1 -18589.969,E2 -18589.969} C_VEL
LIN {X 0,Y 258.113,Z 511.803,A -85,B 0,C 180,E1 -18590.393,E2 -18590.393} C_VEL
LIN {X 0,Y 259.062,Z 513.101,A -85,B 0,C 180,E1 -18590.613,E2 -18590.613} C_VEL
LIN {X 0,Y 267.992,Z 527.463,A -85,B 0,C 180,E1 -18592.651,E2 -18592.651} C_VEL
LIN {X 0,Y 275.667,Z 539.742,A -85,B 0,C 180,E1 -18594.255,E2 -18594.255} C_VEL
LIN {X 0,Y 282.308,Z 548.208,A -85,B 0,C 180,E1 -18595.484,E2 -18595.484} C_VEL
LIN {X 0,Y 292.273,Z 559.211,A -85,B 0,C 180,E1 -18597.143,E2 -18597.143} C_VEL
LIN {X 0,Y 301.407,Z 567.957,A -85,B 0,C 180,E1 -18598.654,E2 -18598.654} C_VEL
LIN {X 0,Y 307.716,Z 574.091,A -85,B 0,C 180,E1 -18599.825,E2 -18599.825} C_VEL
LIN {X 0,Y 315.167,Z 581.075,A -85,B 0,C 180,E1 -18601.341,E2 -18601.341} C_VEL
LIN {X 0,Y 322.827,Z 588.082,A -85,B 0,C 180,E1 -18603.086,E2 -18603.086} C_VEL
LIN {X 0,Y 331.429,Z 595.628,A -85,B 0,C 180,E1 -18605.217,E2 -18605.217} C_VEL
LIN {X 0,Y 336.697,Z 600.079,A -85,B 0,C 180,E1 -18606.618,E2 -18606.618} C_VEL
LIN {X 0,Y 342.915,Z 604.968,A -85,B 0,C 180,E1 -18608.377,E2 -18608.377} C_VEL
LIN {X 0,Y 349.204,Z 610.236,A -85,B 0,C 180,E1 -18610.324,E2 -18610.324} C_VEL
LIN {X 0,Y 355.477,Z 614.797,A -85,B 0,C 180,E1 -18612.461,E2 -18612.461} C_VEL
LIN {X 0,Y 359.822,Z 618.478,A -85,B 0,C 180,E1 -18614.131,E2 -18614.131} C_VEL
LIN {X 0,Y 364.153,Z 621.353,A -85,B 0,C 180,E1 -18615.95,E2 -18615.95} C_VEL
LIN {X 0,Y 367.143,Z 623.225,A -85,B 0,C 180,E1 -18617.359,E2 -18617.359} C_VEL
LIN {X 0,Y 370.951,Z 626.509,A -85,B 0,C 180,E1 -18619.476,E2 -18619.476} C_VEL
LIN {X 0,Y 373.794,Z 628.424,A -85,B 0,C 180,E1 -18621.349,E2 -18621.349} C_VEL
LIN {X 0,Y 376.487,Z 629.909,A -85,B 0,C 180,E1 -18623.569,E2 -18623.569} C_VEL
LIN {X 0,Y 378.373,Z 630.765,A -85,B 0,C 180,E1 -18625.739,E2 -18625.739} C_VEL
LIN {X 0,Y 379.509,Z 631.185,A -85,B 0,C 180,E1 -18627.877,E2 -18627.877} C_VEL
LIN {X 0,Y 379.784,Z 631.38,A -85,B 0,C 180,E1 -18628.94,E2 -18628.94} C_VEL
LIN {X 0,Y 379.896,Z 631.279,A -85,B 0,C 180,E1 -18630,E2 -18630} C_VEL
LIN {X 0,Y 379.652,Z 631.302,A -85,B 0,C 180,E1 -18631.581,E2 -18631.581} C_VEL
LIN {X 0,Y 379.045,Z 630.942,A -85,B 0,C 180,E1 -18633.189,E2 -18633.189} C_VEL
LIN {X 0,Y 377.525,Z 630.436,A -85,B 0,C 180,E1 -18635.341,E2 -18635.341} C_VEL
LIN {X 0,Y 375.239,Z 629.3,A -85,B 0,C 180,E1 -18637.533,E2 -18637.533} C_VEL
LIN {X 0,Y 372.278,Z 627.425,A -85,B 0,C 180,E1 -18639.693,E2 -18639.693} C_VEL
LIN {X 0,Y 369.301,Z 625.087,A -85,B 0,C 180,E1 -18641.492,E2 -18641.492} C_VEL
LIN {X 0,Y 365.751,Z 622.204,A -85,B 0,C 180,E1 -18643.331,E2 -18643.331} C_VEL
LIN {X 0,Y 361.242,Z 619.503,A -85,B 0,C 180,E1 -18645.295,E2 -18645.295} C_VEL
LIN {X 0,Y 356.202,Z 615.486,A -85,B 0,C 180,E1 -18647.27,E2 -18647.27} C_VEL
LIN {X 0,Y 353.133,Z 613.052,A -85,B 0,C 180,E1 -18648.367,E2 -18648.367} C_VEL
LIN {X 0,Y 347.641,Z 609.015,A -85,B 0,C 180,E1 -18650.171,E2 -18650.171} C_VEL
LIN {X 0,Y 342.494,Z 604.682,A -85,B 0,C 180,E1 -18651.744,E2 -18651.744} C_VEL
LIN {X 0,Y 336.583,Z 599.955,A -85,B 0,C 180,E1 -18653.414,E2 -18653.414} C_VEL
LIN {X 0,Y 330.444,Z 594.822,A -85,B 0,C 180,E1 -18655.032,E2 -18655.032} C_VEL
LIN {X 0,Y 322.45,Z 587.724,A -85,B 0,C 180,E1 -18657.004,E2 -18657.004} C_VEL
LIN {X 0,Y 314.235,Z 580.252,A -85,B 0,C 180,E1 -18658.86,E2 -18658.86} C_VEL
LIN {X 0,Y 305.461,Z 572.07,A -85,B 0,C 180,E1 -18660.606,E2 -18660.606} C_VEL
LIN {X 0,Y 296.059,Z 562.822,A -85,B 0,C 180,E1 -18662.256,E2 -18662.256} C_VEL
LIN {X 0,Y 288.622,Z 555.248,A -85,B 0,C 180,E1 -18663.446,E2 -18663.446} C_VEL
LIN {X 0,Y 279.845,Z 545.381,A -85,B 0,C 180,E1 -18664.953,E2 -18664.953} C_VEL
LIN {X 0,Y 272.099,Z 534.357,A -85,B 0,C 180,E1 -18666.465,E2 -18666.465} C_VEL
LIN {X 0,Y 263.085,Z 519.456,A -85,B 0,C 180,E1 -18668.449,E2 -18668.449} C_VEL
LIN {X 0,Y 258.234,Z 511.931,A -85,B 0,C 180,E1 -18669.581,E2 -18669.581} C_VEL
LIN {X 0,Y 256.53,Z 509.305,A -85,B 0,C 180,E1 -18670.004,E2 -18670.004} C_VEL
LIN {X 0,Y 256.182,Z 508.003,A -85,B 0,C 180,E1 -18670.295,E2 -18670.295} C_VEL
LIN {X 0,Y 256.107,Z 507.67,A -85,B 0,C 180,E1 -18671.192,E2 -18671.192} C_VEL
LIN {X 0,Y 256.111,Z 507.66,A -85,B 0,C 180,E1 -18674.483,E2 -18674.483} C_VEL
LIN {X 0,Y 256.127,Z 507.698,A -85,B 0,C 180,E1 -18677.804,E2 -18677.804} C_VEL
LIN {X 0,Y 256.103,Z 507.706,A -85,B 0,C 180,E1 -18680.865,E2 -18680.865} C_VEL
LIN {X 0,Y 256.115,Z 507.691,A -85,B 0,C 180,E1 -18684.813,E2 -18684.813} C_VEL
LIN {X 0,Y 256.087,Z 507.69,A -85,B 0,C 180,E1 -18688.573,E2 -18688.573} C_VEL
LIN {X 0,Y 256.136,Z 507.704,A -85,B 0,C 180,E1 -18692.197,E2 -18692.197} C_VEL
LIN {X 0,Y 256.161,Z 507.672,A -85,B 0,C 180,E1 -18695.699,E2 -18695.699} C_VEL
LIN {X 0,Y 256.161,Z 507.701,A -85,B 0,C 180,E1 -18699.105,E2 -18699.105} C_VEL
LIN {X 0,Y 256.273,Z 507.666,A -85,B 0,C 180,E1 -18704.084,E2 -18704.084} C_VEL
LIN {X 0,Y 256.287,Z 507.681,A -85,B 0,C 180,E1 -18707.328,E2 -18707.328} C_VEL
LIN {X 0,Y 256.51,Z 507.641,A -85,B 0,C 180,E1 -18712.127,E2 -18712.127} C_VEL
LIN {X 0,Y 256.494,Z 507.625,A -85,B 0,C 180,E1 -18716.859,E2 -18716.859} C_VEL
LIN {X 0,Y 256.759,Z 507.608,A -85,B 0,C 180,E1 -18720.001,E2 -18720.001} C_VEL
LIN {X 0,Y 256.494,Z 507.651,A -85,B 0,C 180,E1 -18723.142,E2 -18723.142} C_VEL
LIN {X 0,Y 256.532,Z 507.639,A -85,B 0,C 180,E1 -18727.874,E2 -18727.874} C_VEL
LIN {X 0,Y 256.304,Z 507.676,A -85,B 0,C 180,E1 -18731.067,E2 -18731.067} C_VEL
LIN {X 0,Y 256.29,Z 507.678,A -85,B 0,C 180,E1 -18735.916,E2 -18735.916} C_VEL
LIN {X 0,Y 256.158,Z 507.671,A -85,B 0,C 180,E1 -18740.897,E2 -18740.897} C_VEL
LIN {X 0,Y 256.167,Z 507.694,A -85,B 0,C 180,E1 -18745.131,E2 -18745.131} C_VEL
LIN {X 0,Y 256.1,Z 507.707,A -85,B 0,C 180,E1 -18749.602,E2 -18749.602} C_VEL
LIN {X 0,Y 256.083,Z 507.689,A -85,B 0,C 180,E1 -18753.291,E2 -18753.291} C_VEL
LIN {X 0,Y 256.137,Z 507.692,A -85,B 0,C 180,E1 -18757.279,E2 -18757.279} C_VEL
LIN {X 0,Y 256.081,Z 507.704,A -85,B 0,C 180,E1 -18761.199,E2 -18761.199} C_VEL
LIN {X 0,Y 256.051,Z 507.709,A -85,B 0,C 180,E1 -18763.824,E2 -18763.824} C_VEL
LIN {X 0,Y 255.466,Z 508.21,A -85,B 0,C 180,E1 -18764.692,E2 -18764.692} C_VEL
LIN {X 0,Y 253.649,Z 509.968,A -85,B 0,C 180,E1 -18765.76,E2 -18765.76} C_VEL
LIN {X 0,Y 250.999,Z 513.655,A -85,B 0,C 180,E1 -18767.318,E2 -18767.318} C_VEL
LIN {X 0,Y 250.771,Z 515.428,A -85,B 0,C 180,E1 -18768.152,E2 -18768.152} C_VEL
LIN {X 0,Y 251.194,Z 517.005,A -85,B 0,C 180,E1 -18768.817,E2 -18768.817} C_VEL
LIN {X 0,Y 253.561,Z 521.361,A -85,B 0,C 180,E1 -18769.486,E2 -18769.486} C_VEL
LIN {X 0,Y 261.308,Z 535.988,A -85,B 0,C 180,E1 -18771.417,E2 -18771.417} C_VEL
LIN {X 0,Y 268.201,Z 550.654,A -85,B 0,C 180,E1 -18773.056,E2 -18773.056} C_VEL
LIN {X 0,Y 272.537,Z 561.215,A -85,B 0,C 180,E1 -18774.07,E2 -18774.07} C_VEL
LIN {X 0,Y 275.551,Z 578.378,A -85,B 0,C 180,E1 -18775.055,E2 -18775.055} C_VEL
LIN {X 0,Y 272.422,Z 652.881,A -85,B 0,C 180,E1 -18776.965,E2 -18776.965} C_VEL
LIN {X 0,Y 271.482,Z 664.035,A -85,B 0,C 180,E1 -18777.4,E2 -18777.4} C_VEL
LIN {X 0,Y 270.194,Z 675.024,A -85,B 0,C 180,E1 -18777.997,E2 -18777.997} C_VEL
LIN {X 0,Y 268.706,Z 684.814,A -85,B 0,C 180,E1 -18778.68,E2 -18778.68} C_VEL
LIN {X 0,Y 267,Z 694.783,A -85,B 0,C 180,E1 -18779.556,E2 -18779.556} C_VEL
LIN {X 0,Y 265.03,Z 704.7,A -85,B 0,C 180,E1 -18780.622,E2 -18780.622} C_VEL
LIN {X 0,Y 262.775,Z 714.891,A -85,B 0,C 180,E1 -18781.958,E2 -18781.958} C_VEL
LIN {X 0,Y 260.755,Z 723.845,A -85,B 0,C 180,E1 -18783.38,E2 -18783.38} C_VEL
LIN {X 0,Y 258.287,Z 732.862,A -85,B 0,C 180,E1 -18785.055,E2 -18785.055} C_VEL
LIN {X 0,Y 256.315,Z 739.834,A -85,B 0,C 180,E1 -18786.574,E2 -18786.574} C_VEL
LIN {X 0,Y 254.196,Z 747.357,A -85,B 0,C 180,E1 -18788.511,E2 -18788.511} C_VEL
LIN {X 0,Y 252.375,Z 753.832,A -85,B 0,C 180,E1 -18790.478,E2 -18790.478} C_VEL
LIN {X 0,Y 251.03,Z 758.625,A -85,B 0,C 180,E1 -18792.156,E2 -18792.156} C_VEL
LIN {X 0,Y 249.67,Z 764.196,A -85,B 0,C 180,E1 -18794.49,E2 -18794.49} C_VEL
LIN {X 0,Y 248.104,Z 770.258,A -85,B 0,C 180,E1 -18797.734,E2 -18797.734} C_VEL
LIN {X 0,Y 247.45,Z 773.809,A -85,B 0,C 180,E1 -18800.189,E2 -18800.189} C_VEL
LIN {X 0,Y 247.162,Z 775.753,A -85,B 0,C 180,E1 -18801.827,E2 -18801.827} C_VEL
LIN {X 0,Y 246.884,Z 778.445,A -85,B 0,C 180,E1 -18805.101,E2 -18805.101} C_VEL
LIN {X 0,Y 246.925,Z 779.743,A -85,B 0,C 180,E1 -18808.369,E2 -18808.369} C_VEL
LIN {X 0,Y 246.984,Z 779.997,A -85,B 0,C 180,E1 -18810,E2 -18810} C_VEL
LIN {X 0,Y 246.852,Z 779.265,A -85,B 0,C 180,E1 -18813.264,E2 -18813.264} C_VEL
LIN {X 0,Y 246.884,Z 778.445,A -85,B 0,C 180,E1 -18814.899,E2 -18814.899} C_VEL
LIN {X 0,Y 247.162,Z 775.753,A -85,B 0,C 180,E1 -18818.173,E2 -18818.173} C_VEL
LIN {X 0,Y 247.65,Z 772.792,A -85,B 0,C 180,E1 -18820.63,E2 -18820.63} C_VEL
LIN {X 0,Y 248.42,Z 768.959,A -85,B 0,C 180,E1 -18823.081,E2 -18823.081} C_VEL
LIN {X 0,Y 249.659,Z 764.196,A -85,B 0,C 180,E1 -18825.511,E2 -18825.511} C_VEL
LIN {X 0,Y 251.419,Z 757.246,A -85,B 0,C 180,E1 -18828.329,E2 -18828.329} C_VEL
LIN {X 0,Y 253.457,Z 750.033,A -85,B 0,C 180,E1 -18830.703,E2 -18830.703} C_VEL
LIN {X 0,Y 255.454,Z 742.958,A -85,B 0,C 180,E1 -18832.653,E2 -18832.653} C_VEL
LIN {X 0,Y 257.225,Z 736.496,A -85,B 0,C 180,E1 -18834.194,E2 -18834.194} C_VEL
LIN {X 0,Y 259.885,Z 727.022,A -85,B 0,C 180,E1 -18836.068,E2 -18836.068} C_VEL
LIN {X 0,Y 262.04,Z 718.659,A -85,B 0,C 180,E1 -18837.468,E2 -18837.468} C_VEL
LIN {X 0,Y 264.124,Z 709.094,A -85,B 0,C 180,E1 -18838.834,E2 -18838.834} C_VEL
LIN {X 0,Y 266.34,Z 698.29,A -85,B 0,C 180,E1 -18840.089,E2 -18840.089} C_VEL
LIN {X 0,Y 268.188,Z 688.034,A -85,B 0,C 180,E1 -18841.058,E2 -18841.058} C_VEL
LIN {X 0,Y 270.005,Z 676.384,A -85,B 0,C 180,E1 -18841.918,E2 -18841.918} C_VEL
LIN {X 0,Y 271.292,Z 665.859,A -85,B 0,C 180,E1 -18842.516,E2 -18842.516} C_VEL
LIN {X 0,Y 272.229,Z 655.068,A -85,B 0,C 180,E1 -18842.969,E2 -18842.969} C_VEL
LIN {X 0,Y 273.509,Z 630.084,A -85,B 0,C 180,E1 -18843.634,E2 -18843.634} C_VEL
LIN {X 0,Y 275.459,Z 577.414,A -85,B 0,C 180,E1 -18844.988,E2 -18844.988} C_VEL
LIN {X 0,Y 272.373,Z 560.653,A -85,B 0,C 180,E1 -18845.973,E2 -18845.973} C_VEL
LIN {X 0,Y 265.931,Z 545.606,A -85,B 0,C 180,E1 -18847.478,E2 -18847.478} C_VEL
LIN {X 0,Y 259.622,Z 532.749,A -85,B 0,C 180,E1 -18848.991,E2 -18848.991} C_VEL
LIN {X 0,Y 253.135,Z 520.736,A -85,B 0,C 180,E1 -18850.618,E2 -18850.618} C_VEL
LIN {X 0,Y 251.131,Z 516.821,A -85,B 0,C 180,E1 -18851.228,E2 -18851.228} C_VEL
LIN {X 0,Y 249.368,Z 510.034,A -85,B 0,C 180,E1 -18854.794,E2 -18854.794} C_VEL
LIN {X 0,Y 249.021,Z 508.589,A -85,B 0,C 180,E1 -18855.754,E2 -18855.754} C_VEL
LIN {X 0,Y 249.046,Z 508.588,A -85,B 0,C 180,E1 -18859.633,E2 -18859.633} C_VEL
LIN {X 0,Y 249.072,Z 508.581,A -85,B 0,C 180,E1 -18863.661,E2 -18863.661} C_VEL
LIN {X 0,Y 249.037,Z 508.57,A -85,B 0,C 180,E1 -18867.844,E2 -18867.844} C_VEL
LIN {X 0,Y 249.082,Z 508.566,A -85,B 0,C 180,E1 -18871.336,E2 -18871.336} C_VEL
LIN {X 0,Y 249.131,Z 508.571,A -85,B 0,C 180,E1 -18874.966,E2 -18874.966} C_VEL
LIN {X 0,Y 249.09,Z 508.553,A -85,B 0,C 180,E1 -18878.601,E2 -18878.601} C_VEL
LIN {X 0,Y 249.238,Z 508.56,A -85,B 0,C 180,E1 -18883.621,E2 -18883.621} C_VEL
LIN {X 0,Y 249.247,Z 508.547,A -85,B 0,C 180,E1 -18888.616,E2 -18888.616} C_VEL
LIN {X 0,Y 249.475,Z 508.521,A -85,B 0,C 180,E1 -18891.902,E2 -18891.902} C_VEL
LIN {X 0,Y 249.43,Z 508.528,A -85,B 0,C 180,E1 -18896.769,E2 -18896.769} C_VEL
LIN {X 0,Y 249.722,Z 508.483,A -85,B 0,C 180,E1 -18899.999,E2 -18899.999} C_VEL
LIN {X 0,Y 249.429,Z 508.505,A -85,B 0,C 180,E1 -18903.23,E2 -18903.23} C_VEL
LIN {X 0,Y 249.435,Z 508.531,A -85,B 0,C 180,E1 -18906.711,E2 -18906.711} C_VEL
LIN {X 0,Y 249.337,Z 508.514,A -85,B 0,C 180,E1 -18909.736,E2 -18909.736} C_VEL
LIN {X 0,Y 249.192,Z 508.565,A -85,B 0,C 180,E1 -18914.703,E2 -18914.703} C_VEL
LIN {X 0,Y 249.129,Z 508.546,A -85,B 0,C 180,E1 -18918.077,E2 -18918.077} C_VEL
LIN {X 0,Y 249.081,Z 508.581,A -85,B 0,C 180,E1 -18921.518,E2 -18921.518} C_VEL
LIN {X 0,Y 249.125,Z 508.555,A -85,B 0,C 180,E1 -18925.482,E2 -18925.482} C_VEL
LIN {X 0,Y 249.078,Z 508.569,A -85,B 0,C 180,E1 -18928.993,E2 -18928.993} C_VEL
LIN {X 0,Y 249.03,Z 508.581,A -85,B 0,C 180,E1 -18932.425,E2 -18932.425} C_VEL
LIN {X 0,Y 249.069,Z 508.565,A -85,B 0,C 180,E1 -18936.338,E2 -18936.338} C_VEL
LIN {X 0,Y 249.072,Z 508.568,A -85,B 0,C 180,E1 -18940.464,E2 -18940.464} C_VEL
LIN {X 0,Y 249.057,Z 508.548,A -85,B 0,C 180,E1 -18944.866,E2 -18944.866} C_VEL
LIN {X 0,Y 249.102,Z 508.7,A -85,B 0,C 180,E1 -18948.197,E2 -18948.197} C_VEL
LIN {X 0,Y 249.318,Z 509.734,A -85,B 0,C 180,E1 -18948.581,E2 -18948.581} C_VEL
LIN {X 0,Y 250.9,Z 512.523,A -85,B 0,C 180,E1 -18949.033,E2 -18949.033} C_VEL
LIN {X 0,Y 252.013,Z 513.878,A -85,B 0,C 180,E1 -18949.304,E2 -18949.304} C_VEL
LIN {X 0,Y 260.576,Z 527.315,A -85,B 0,C 180,E1 -18951.382,E2 -18951.382} C_VEL
LIN {X 0,Y 270.793,Z 544.072,A -85,B 0,C 180,E1 -18953.644,E2 -18953.644} C_VEL
LIN {X 0,Y 277.656,Z 552.995,A -85,B 0,C 180,E1 -18954.965,E2 -18954.965} C_VEL
LIN {X 0,Y 287.837,Z 564.339,A -85,B 0,C 180,E1 -18956.717,E2 -18956.717} C_VEL
LIN {X 0,Y 298.165,Z 574.228,A -85,B 0,C 180,E1 -18958.376,E2 -18958.376} C_VEL
LIN {X 0,Y 305.57,Z 581.127,A -85,B 0,C 180,E1 -18959.694,E2 -18959.694} C_VEL
LIN {X 0,Y 312.255,Z 587.289,A -85,B 0,C 180,E1 -18961.009,E2 -18961.009} C_VEL
LIN {X 0,Y 319.913,Z 594.167,A -85,B 0,C 180,E1 -18962.691,E2 -18962.691} C_VEL
LIN {X 0,Y 328.871,Z 601.931,A -85,B 0,C 180,E1 -18964.863,E2 -18964.863} C_VEL
LIN {X 0,Y 334.535,Z 606.635,A -85,B 0,C 180,E1 -18966.336,E2 -18966.336} C_VEL
LIN {X 0,Y 340.876,Z 611.533,A -85,B 0,C 180,E1 -18968.09,E2 -18968.09} C_VEL
LIN {X 0,Y 347.361,Z 616.914,A -85,B 0,C 180,E1 -18970.069,E2 -18970.069} C_VEL
LIN {X 0,Y 353.943,Z 621.677,A -85,B 0,C 180,E1 -18972.264,E2 -18972.264} C_VEL
LIN {X 0,Y 358.739,Z 625.604,A -85,B 0,C 180,E1 -18974.082,E2 -18974.082} C_VEL
LIN {X 0,Y 363.454,Z 628.6,A -85,B 0,C 180,E1 -18976.056,E2 -18976.056} C_VEL
LIN {X 0,Y 365.772,Z 630.045,A -85,B 0,C 180,E1 -18977.137,E2 -18977.137} C_VEL
LIN {X 0,Y 369.678,Z 633.361,A -85,B 0,C 180,E1 -18979.26,E2 -18979.26} C_VEL
LIN {X 0,Y 372.877,Z 635.465,A -85,B 0,C 180,E1 -18981.328,E2 -18981.328} C_VEL
LIN {X 0,Y 375.594,Z 636.947,A -85,B 0,C 180,E1 -18983.554,E2 -18983.554} C_VEL
LIN {X 0,Y 377.496,Z 637.81,A -85,B 0,C 180,E1 -18985.729,E2 -18985.729} C_VEL
LIN {X 0,Y 378.641,Z 638.233,A -85,B 0,C 180,E1 -18987.873,E2 -18987.873} C_VEL
LIN {X 0,Y 378.918,Z 638.426,A -85,B 0,C 180,E1 -18988.937,E2 -18988.937} C_VEL
LIN {X 0,Y 379.03,Z 638.326,A -85,B 0,C 180,E1 -18990,E2 -18990} C_VEL
LIN {X 0,Y 378.918,Z 638.427,A -85,B 0,C 180,E1 -18991.063,E2 -18991.063} C_VEL
LIN {X 0,Y 378.173,Z 637.988,A -85,B 0,C 180,E1 -18993.196,E2 -18993.196} C_VEL
LIN {X 0,Y 376.641,Z 637.48,A -85,B 0,C 180,E1 -18995.353,E2 -18995.353} C_VEL
LIN {X 0,Y 374.337,Z 636.325,A -85,B 0,C 180,E1 -18997.552,E2 -18997.552} C_VEL
LIN {X 0,Y 371.34,Z 634.504,A -85,B 0,C 180,E1 -18999.717,E2 -18999.717} C_VEL
LIN {X 0,Y 368.317,Z 632.22,A -85,B 0,C 180,E1 -19001.523,E2 -19001.523} C_VEL
LIN {X 0,Y 364.732,Z 629.259,A -85,B 0,C 180,E1 -19003.369,E2 -19003.369} C_VEL
LIN {X 0,Y 360.169,Z 626.58,A -85,B 0,C 180,E1 -19005.341,E2 -19005.341} C_VEL
LIN {X 0,Y 355.22,Z 622.798,A -85,B 0,C 180,E1 -19007.263,E2 -19007.263} C_VEL
LIN {X 0,Y 351.498,Z 619.826,A -85,B 0,C 180,E1 -19008.587,E2 -19008.587} C_VEL
LIN {X 0,Y 346.078,Z 615.909,A -85,B 0,C 180,E1 -19010.34,E2 -19010.34} C_VEL
LIN {X 0,Y 339.709,Z 610.731,A -85,B 0,C 180,E1 -19012.237,E2 -19012.237} C_VEL
LIN {X 0,Y 333.677,Z 605.86,A -85,B 0,C 180,E1 -19013.897,E2 -19013.897} C_VEL
LIN {X 0,Y 325.268,Z 598.875,A -85,B 0,C 180,E1 -19016.031,E2 -19016.031} C_VEL
LIN {X 0,Y 317.927,Z 592.474,A -85,B 0,C 180,E1 -19017.758,E2 -19017.758} C_VEL
LIN {X 0,Y 310.957,Z 586.17,A -85,B 0,C 180,E1 -19019.25,E2 -19019.25} C_VEL
LIN {X 0,Y 302.219,Z 578.166,A -85,B 0,C 180,E1 -19020.912,E2 -19020.912} C_VEL
LIN {X 0,Y 292.714,Z 569.08,A -85,B 0,C 180,E1 -19022.513,E2 -19022.513} C_VEL
LIN {X 0,Y 280.503,Z 556.476,A -85,B 0,C 180,E1 -19024.52,E2 -19024.52} C_VEL
LIN {X 0,Y 272.727,Z 546.676,A -85,B 0,C 180,E1 -19025.972,E2 -19025.972} C_VEL
LIN {X 0,Y 266.09,Z 536.745,A -85,B 0,C 180,E1 -19027.354,E2 -19027.354} C_VEL
LIN {X 0,Y 258.244,Z 523.635,A -85,B 0,C 180,E1 -19029.165,E2 -19029.165} C_VEL
LIN {X 0,Y 253.634,Z 516.516,A -85,B 0,C 180,E1 -19030.284,E2 -19030.284} C_VEL
LIN {X 0,Y 251.266,Z 512.852,A -85,B 0,C 180,E1 -19030.882,E2 -19030.882} C_VEL
LIN {X 0,Y 249.548,Z 510.327,A -85,B 0,C 180,E1 -19031.33,E2 -19031.33} C_VEL
LIN {X 0,Y 249.116,Z 508.901,A -85,B 0,C 180,E1 -19031.645,E2 -19031.645} C_VEL
LIN {X 0,Y 249.074,Z 508.529,A -85,B 0,C 180,E1 -19032.624,E2 -19032.624} C_VEL
LIN {X 0,Y 249.073,Z 508.583,A -85,B 0,C 180,E1 -19037.376,E2 -19037.376} C_VEL
LIN {X 0,Y 249.047,Z 508.59,A -85,B 0,C 180,E1 -19041.624,E2 -19041.624} C_VEL
LIN {X 0,Y 249.056,Z 508.579,A -85,B 0,C 180,E1 -19045.642,E2 -19045.642} C_VEL
LIN {X 0,Y 249.046,Z 508.562,A -85,B 0,C 180,E1 -19049.473,E2 -19049.473} C_VEL
LIN {X 0,Y 249.068,Z 508.583,A -85,B 0,C 180,E1 -19053.163,E2 -19053.163} C_VEL
LIN {X 0,Y 249.073,Z 508.559,A -85,B 0,C 180,E1 -19056.733,E2 -19056.733} C_VEL
LIN {X 0,Y 249.104,Z 508.572,A -85,B 0,C 180,E1 -19060.212,E2 -19060.212} C_VEL
LIN {X 0,Y 249.217,Z 508.538,A -85,B 0,C 180,E1 -19063.621,E2 -19063.621} C_VEL
LIN {X 0,Y 249.238,Z 508.537,A -85,B 0,C 180,E1 -19068.617,E2 -19068.617} C_VEL
LIN {X 0,Y 249.449,Z 508.515,A -85,B 0,C 180,E1 -19071.903,E2 -19071.903} C_VEL
LIN {X 0,Y 249.293,Z 508.548,A -85,B 0,C 180,E1 -19075.149,E2 -19075.149} C_VEL
LIN {X 0,Y 249.67,Z 508.47,A -85,B 0,C 180,E1 -19078.388,E2 -19078.388} C_VEL
LIN {X 0,Y 249.67,Z 508.506,A -85,B 0,C 180,E1 -19081.614,E2 -19081.614} C_VEL
LIN {X 0,Y 249.454,Z 508.5,A -85,B 0,C 180,E1 -19086.471,E2 -19086.471} C_VEL
LIN {X 0,Y 249.384,Z 508.546,A -85,B 0,C 180,E1 -19089.736,E2 -19089.736} C_VEL
LIN {X 0,Y 249.196,Z 508.54,A -85,B 0,C 180,E1 -19094.705,E2 -19094.705} C_VEL
LIN {X 0,Y 249.133,Z 508.571,A -85,B 0,C 180,E1 -19098.078,E2 -19098.078} C_VEL
LIN {X 0,Y 249.08,Z 508.555,A -85,B 0,C 180,E1 -19101.519,E2 -19101.519} C_VEL
LIN {X 0,Y 249.113,Z 508.566,A -85,B 0,C 180,E1 -19105.476,E2 -19105.476} C_VEL
LIN {X 0,Y 249.07,Z 508.573,A -85,B 0,C 180,E1 -19108.99,E2 -19108.99} C_VEL
LIN {X 0,Y 249.033,Z 508.569,A -85,B 0,C 180,E1 -19112.426,E2 -19112.426} C_VEL
LIN {X 0,Y 249.072,Z 508.581,A -85,B 0,C 180,E1 -19116.339,E2 -19116.339} C_VEL
LIN {X 0,Y 249.043,Z 508.589,A -85,B 0,C 180,E1 -19120.472,E2 -19120.472} C_VEL
LIN {X 0,Y 249.045,Z 508.751,A -85,B 0,C 180,E1 -19124.449,E2 -19124.449} C_VEL
LIN {X 0,Y 250.771,Z 515.428,A -85,B 0,C 180,E1 -19128.152,E2 -19128.152} C_VEL
LIN {X 0,Y 251.461,Z 517.209,A -85,B 0,C 180,E1 -19128.753,E2 -19128.753} C_VEL
LIN {X 0,Y 252.969,Z 520.847,A -85,B 0,C 180,E1 -19129.354,E2 -19129.354} C_VEL
LIN {X 0,Y 254.846,Z 527.497,A -85,B 0,C 180,E1 -19129.952,E2 -19129.952} C_VEL
LIN {X 0,Y 256.997,Z 539.519,A -85,B 0,C 180,E1 -19130.765,E2 -19130.765} C_VEL
LIN {X 0,Y 258.089,Z 543.305,A -85,B 0,C 180,E1 -19131.105,E2 -19131.105} C_VEL
LIN {X 0,Y 265.387,Z 559.699,A -85,B 0,C 180,E1 -19132.901,E2 -19132.901} C_VEL
LIN {X 0,Y 267.175,Z 564.653,A -85,B 0,C 180,E1 -19133.351,E2 -19133.351} C_VEL
LIN {X 0,Y 269.679,Z 579.094,A -85,B 0,C 180,E1 -19134.208,E2 -19134.208} C_VEL
LIN {X 0,Y 266.558,Z 651.828,A -85,B 0,C 180,E1 -19136.104,E2 -19136.104} C_VEL
LIN {X 0,Y 265.636,Z 662.926,A -85,B 0,C 180,E1 -19136.533,E2 -19136.533} C_VEL
LIN {X 0,Y 264.396,Z 673.466,A -85,B 0,C 180,E1 -19137.095,E2 -19137.095} C_VEL
LIN {X 0,Y 262.666,Z 684.615,A -85,B 0,C 180,E1 -19137.875,E2 -19137.875} C_VEL
LIN {X 0,Y 260.887,Z 694.584,A -85,B 0,C 180,E1 -19138.764,E2 -19138.764} C_VEL
LIN {X 0,Y 258.863,Z 704.502,A -85,B 0,C 180,E1 -19139.851,E2 -19139.851} C_VEL
LIN {X 0,Y 256.576,Z 714.484,A -85,B 0,C 180,E1 -19141.181,E2 -19141.181} C_VEL
LIN {X 0,Y 254.378,Z 723.646,A -85,B 0,C 180,E1 -19142.658,E2 -19142.658} C_VEL
LIN {X 0,Y 251.839,Z 732.663,A -85,B 0,C 180,E1 -19144.371,E2 -19144.371} C_VEL
LIN {X 0,Y 249.755,Z 739.634,A -85,B 0,C 180,E1 -19145.92,E2 -19145.92} C_VEL
LIN {X 0,Y 247.564,Z 747.158,A -85,B 0,C 180,E1 -19147.905,E2 -19147.905} C_VEL
LIN {X 0,Y 245.309,Z 754.771,A -85,B 0,C 180,E1 -19150.329,E2 -19150.329} C_VEL
LIN {X 0,Y 243.73,Z 760.499,A -85,B 0,C 180,E1 -19152.522,E2 -19152.522} C_VEL
LIN {X 0,Y 242.337,Z 765.613,A -85,B 0,C 180,E1 -19154.87,E2 -19154.87} C_VEL
LIN {X 0,Y 241.126,Z 770.059,A -85,B 0,C 180,E1 -19157.374,E2 -19157.374} C_VEL
LIN {X 0,Y 240.419,Z 773.61,A -85,B 0,C 180,E1 -19159.899,E2 -19159.899} C_VEL
LIN {X 0,Y 240.093,Z 775.554,A -85,B 0,C 180,E1 -19161.584,E2 -19161.584} C_VEL
LIN {X 0,Y 239.792,Z 778.37,A -85,B 0,C 180,E1 -19165.209,E2 -19165.209} C_VEL
LIN {X 0,Y 239.834,Z 779.545,A -85,B 0,C 180,E1 -19168.321,E2 -19168.321} C_VEL
LIN {X 0,Y 239.893,Z 779.799,A -85,B 0,C 180,E1 -19170,E2 -19170} C_VEL
LIN {X 0,Y 239.759,Z 779.067,A -85,B 0,C 180,E1 -19173.361,E2 -19173.361} C_VEL
LIN {X 0,Y 239.802,Z 778.247,A -85,B 0,C 180,E1 -19175.044,E2 -19175.044} C_VEL
LIN {X 0,Y 240.093,Z 775.554,A -85,B 0,C 180,E1 -19178.416,E2 -19178.416} C_VEL
LIN {X 0,Y 240.628,Z 772.592,A -85,B 0,C 180,E1 -19180.943,E2 -19180.943} C_VEL
LIN {X 0,Y 241.48,Z 768.761,A -85,B 0,C 180,E1 -19183.463,E2 -19183.463} C_VEL
LIN {X 0,Y 242.762,Z 763.996,A -85,B 0,C 180,E1 -19185.963,E2 -19185.963} C_VEL
LIN {X 0,Y 244.64,Z 757.047,A -85,B 0,C 180,E1 -19188.855,E2 -19188.855} C_VEL
LIN {X 0,Y 246.768,Z 749.833,A -85,B 0,C 180,E1 -19191.292,E2 -19191.292} C_VEL
LIN {X 0,Y 248.883,Z 742.759,A -85,B 0,C 180,E1 -19193.286,E2 -19193.286} C_VEL
LIN {X 0,Y 250.743,Z 736.297,A -85,B 0,C 180,E1 -19194.861,E2 -19194.861} C_VEL
LIN {X 0,Y 253.508,Z 726.823,A -85,B 0,C 180,E1 -19196.775,E2 -19196.775} C_VEL
LIN {X 0,Y 255.98,Z 717.325,A -85,B 0,C 180,E1 -19198.38,E2 -19198.38} C_VEL
LIN {X 0,Y 258.23,Z 707.431,A -85,B 0,C 180,E1 -19199.781,E2 -19199.781} C_VEL
LIN {X 0,Y 260.201,Z 698.091,A -85,B 0,C 180,E1 -19200.876,E2 -19200.876} C_VEL
LIN {X 0,Y 262.133,Z 687.836,A -85,B 0,C 180,E1 -19201.859,E2 -19201.859} C_VEL
LIN {X 0,Y 263.808,Z 677.545,A -85,B 0,C 180,E1 -19202.647,E2 -19202.647} C_VEL
LIN {X 0,Y 265.339,Z 665.661,A -85,B 0,C 180,E1 -19203.339,E2 -19203.339} C_VEL
LIN {X 0,Y 266.383,Z 653.893,A -85,B 0,C 180,E1 -19203.829,E2 -19203.829} C_VEL
LIN {X 0,Y 267.749,Z 626.709,A -85,B 0,C 180,E1 -19204.559,E2 -19204.559} C_VEL
LIN {X 0,Y 269.621,Z 578.455,A -85,B 0,C 180,E1 -19205.822,E2 -19205.822} C_VEL
LIN {X 0,Y 266.903,Z 563.549,A -85,B 0,C 180,E1 -19206.728,E2 -19206.728} C_VEL
LIN {X 0,Y 260.982,Z 549.576,A -85,B 0,C 180,E1 -19208.174,E2 -19208.174} C_VEL
LIN {X 0,Y 255.057,Z 537.275,A -85,B 0,C 180,E1 -19209.658,E2 -19209.658} C_VEL
LIN {X 0,Y 248.485,Z 525.073,A -85,B 0,C 180,E1 -19211.375,E2 -19211.375} C_VEL
LIN {X 0,Y 245.756,Z 520.303,A -85,B 0,C 180,E1 -19212.117,E2 -19212.117} C_VEL
LIN {X 0,Y 243.806,Z 516.515,A -85,B 0,C 180,E1 -19212.762,E2 -19212.762} C_VEL
LIN {X 0,Y 242.005,Z 509.546,A -85,B 0,C 180,E1 -19216.703,E2 -19216.703} C_VEL
LIN {X 0,Y 242.016,Z 509.448,A -85,B 0,C 180,E1 -19221.632,E2 -19221.632} C_VEL
LIN {X 0,Y 242.035,Z 509.462,A -85,B 0,C 180,E1 -19224.496,E2 -19224.496} C_VEL
LIN {X 0,Y 241.972,Z 509.457,A -85,B 0,C 180,E1 -19228.479,E2 -19228.479} C_VEL
LIN {X 0,Y 241.996,Z 509.439,A -85,B 0,C 180,E1 -19232.31,E2 -19232.31} C_VEL
LIN {X 0,Y 242.037,Z 509.461,A -85,B 0,C 180,E1 -19236.013,E2 -19236.013} C_VEL
LIN {X 0,Y 242.031,Z 509.43,A -85,B 0,C 180,E1 -19239.607,E2 -19239.607} C_VEL
LIN {X 0,Y 242.16,Z 509.444,A -85,B 0,C 180,E1 -19243.277,E2 -19243.277} C_VEL
LIN {X 0,Y 242.181,Z 509.42,A -85,B 0,C 180,E1 -19248.279,E2 -19248.279} C_VEL
LIN {X 0,Y 242.422,Z 509.404,A -85,B 0,C 180,E1 -19251.665,E2 -19251.665} C_VEL
LIN {X 0,Y 242.252,Z 509.396,A -85,B 0,C 180,E1 -19255.006,E2 -19255.006} C_VEL
LIN {X 0,Y 242.631,Z 509.383,A -85,B 0,C 180,E1 -19258.339,E2 -19258.339} C_VEL
LIN {X 0,Y 242.63,Z 509.346,A -85,B 0,C 180,E1 -19261.659,E2 -19261.659} C_VEL
LIN {X 0,Y 242.416,Z 509.41,A -85,B 0,C 180,E1 -19266.683,E2 -19266.683} C_VEL
LIN {X 0,Y 242.262,Z 509.395,A -85,B 0,C 180,E1 -19270.023,E2 -19270.023} C_VEL
LIN {X 0,Y 242.151,Z 509.435,A -85,B 0,C 180,E1 -19275.141,E2 -19275.141} C_VEL
LIN {X 0,Y 242.065,Z 509.43,A -85,B 0,C 180,E1 -19278.624,E2 -19278.624} C_VEL
LIN {X 0,Y 242.007,Z 509.454,A -85,B 0,C 180,E1 -19282.18,E2 -19282.18} C_VEL
LIN {X 0,Y 242.061,Z 509.438,A -85,B 0,C 180,E1 -19285.838,E2 -19285.838} C_VEL
LIN {X 0,Y 242.025,Z 509.44,A -85,B 0,C 180,E1 -19289.58,E2 -19289.58} C_VEL
LIN {X 0,Y 241.986,Z 509.469,A -85,B 0,C 180,E1 -19293.491,E2 -19293.491} C_VEL
LIN {X 0,Y 242.006,Z 509.456,A -85,B 0,C 180,E1 -19297.578,E2 -19297.578} C_VEL
LIN {X 0,Y 241.99,Z 509.455,A -85,B 0,C 180,E1 -19301.91,E2 -19301.91} C_VEL
LIN {X 0,Y 242.002,Z 509.412,A -85,B 0,C 180,E1 -19305.816,E2 -19305.816} C_VEL
LIN {X 0,Y 242.054,Z 509.73,A -85,B 0,C 180,E1 -19306.849,E2 -19306.849} C_VEL
LIN {X 0,Y 242.448,Z 511.054,A -85,B 0,C 180,E1 -19307.192,E2 -19307.192} C_VEL
LIN {X 0,Y 244.153,Z 513.656,A -85,B 0,C 180,E1 -19307.678,E2 -19307.678} C_VEL
LIN {X 0,Y 245.133,Z 514.944,A -85,B 0,C 180,E1 -19307.937,E2 -19307.937} C_VEL
LIN {X 0,Y 247.348,Z 518.265,A -85,B 0,C 180,E1 -19308.528,E2 -19308.528} C_VEL
LIN {X 0,Y 255.829,Z 531.574,A -85,B 0,C 180,E1 -19310.673,E2 -19310.673} C_VEL
LIN {X 0,Y 266.399,Z 549.045,A -85,B 0,C 180,E1 -19313.105,E2 -19313.105} C_VEL
LIN {X 0,Y 273.45,Z 558.282,A -85,B 0,C 180,E1 -19314.507,E2 -19314.507} C_VEL
LIN {X 0,Y 283.973,Z 570.054,A -85,B 0,C 180,E1 -19316.37,E2 -19316.37} C_VEL
LIN {X 0,Y 297.183,Z 582.693,A -85,B 0,C 180,E1 -19318.488,E2 -19318.488} C_VEL
LIN {X 0,Y 306.394,Z 591.025,A -85,B 0,C 180,E1 -19320.134,E2 -19320.134} C_VEL
LIN {X 0,Y 314.893,Z 598.518,A -85,B 0,C 180,E1 -19321.851,E2 -19321.851} C_VEL
LIN {X 0,Y 323.014,Z 605.469,A -85,B 0,C 180,E1 -19323.709,E2 -19323.709} C_VEL
LIN {X 0,Y 331.718,Z 612.656,A -85,B 0,C 180,E1 -19325.888,E2 -19325.888} C_VEL
LIN {X 0,Y 338.144,Z 617.685,A -85,B 0,C 180,E1 -19327.626,E2 -19327.626} C_VEL
LIN {X 0,Y 345.232,Z 623.369,A -85,B 0,C 180,E1 -19329.72,E2 -19329.72} C_VEL
LIN {X 0,Y 350.75,Z 627.156,A -85,B 0,C 180,E1 -19331.497,E2 -19331.497} C_VEL
LIN {X 0,Y 356.042,Z 631.469,A -85,B 0,C 180,E1 -19333.415,E2 -19333.415} C_VEL
LIN {X 0,Y 360.641,Z 634.657,A -85,B 0,C 180,E1 -19335.252,E2 -19335.252} C_VEL
LIN {X 0,Y 364.49,Z 636.936,A -85,B 0,C 180,E1 -19336.959,E2 -19336.959} C_VEL
LIN {X 0,Y 368.546,Z 640.316,A -85,B 0,C 180,E1 -19339.126,E2 -19339.126} C_VEL
LIN {X 0,Y 371.697,Z 642.386,A -85,B 0,C 180,E1 -19341.112,E2 -19341.112} C_VEL
LIN {X 0,Y 374.397,Z 643.851,A -85,B 0,C 180,E1 -19343.239,E2 -19343.239} C_VEL
LIN {X 0,Y 376.344,Z 644.732,A -85,B 0,C 180,E1 -19345.317,E2 -19345.317} C_VEL
LIN {X 0,Y 377.547,Z 645.165,A -85,B 0,C 180,E1 -19347.333,E2 -19347.333} C_VEL
LIN {X 0,Y 378.052,Z 645.472,A -85,B 0,C 180,E1 -19348.935,E2 -19348.935} C_VEL
LIN {X 0,Y 378.167,Z 645.362,A -85,B 0,C 180,E1 -19350,E2 -19350} C_VEL
LIN {X 0,Y 378.052,Z 645.473,A -85,B 0,C 180,E1 -19351.065,E2 -19351.065} C_VEL
LIN {X 0,Y 377.301,Z 645.035,A -85,B 0,C 180,E1 -19353.203,E2 -19353.203} C_VEL
LIN {X 0,Y 375.756,Z 644.524,A -85,B 0,C 180,E1 -19355.366,E2 -19355.366} C_VEL
LIN {X 0,Y 373.431,Z 643.376,A -85,B 0,C 180,E1 -19357.57,E2 -19357.57} C_VEL
LIN {X 0,Y 370.445,Z 641.614,A -85,B 0,C 180,E1 -19359.714,E2 -19359.714} C_VEL
LIN {X 0,Y 367.188,Z 639.221,A -85,B 0,C 180,E1 -19361.635,E2 -19361.635} C_VEL
LIN {X 0,Y 363.398,Z 636.144,A -85,B 0,C 180,E1 -19363.549,E2 -19363.549} C_VEL
LIN {X 0,Y 358.554,Z 633.303,A -85,B 0,C 180,E1 -19365.604,E2 -19365.604} C_VEL
LIN {X 0,Y 353.52,Z 629.506,A -85,B 0,C 180,E1 -19367.521,E2 -19367.521} C_VEL
LIN {X 0,Y 349.301,Z 626.216,A -85,B 0,C 180,E1 -19368.98,E2 -19368.98} C_VEL
LIN {X 0,Y 343.656,Z 622.171,A -85,B 0,C 180,E1 -19370.756,E2 -19370.756} C_VEL
LIN {X 0,Y 338.107,Z 617.656,A -85,B 0,C 180,E1 -19372.384,E2 -19372.384} C_VEL
LIN {X 0,Y 331.833,Z 612.759,A -85,B 0,C 180,E1 -19374.082,E2 -19374.082} C_VEL
LIN {X 0,Y 323.017,Z 605.506,A -85,B 0,C 180,E1 -19376.289,E2 -19376.289} C_VEL
LIN {X 0,Y 315.356,Z 598.921,A -85,B 0,C 180,E1 -19378.05,E2 -19378.05} C_VEL
LIN {X 0,Y 307.383,Z 591.892,A -85,B 0,C 180,E1 -19379.679,E2 -19379.679} C_VEL
LIN {X 0,Y 298.381,Z 583.808,A -85,B 0,C 180,E1 -19381.31,E2 -19381.31} C_VEL
LIN {X 0,Y 287.569,Z 573.478,A -85,B 0,C 180,E1 -19383.051,E2 -19383.051} C_VEL
LIN {X 0,Y 276.982,Z 562.529,A -85,B 0,C 180,E1 -19384.838,E2 -19384.838} C_VEL
LIN {X 0,Y 268.566,Z 552.038,A -85,B 0,C 180,E1 -19386.448,E2 -19386.448} C_VEL
LIN {X 0,Y 261.391,Z 541.164,A -85,B 0,C 180,E1 -19387.999,E2 -19387.999} C_VEL
LIN {X 0,Y 253.42,Z 527.695,A -85,B 0,C 180,E1 -19389.918,E2 -19389.918} C_VEL
LIN {X 0,Y 246.94,Z 517.789,A -85,B 0,C 180,E1 -19391.574,E2 -19391.574} C_VEL
LIN {X 0,Y 244.403,Z 513.888,A -85,B 0,C 180,E1 -19392.26,E2 -19392.26} C_VEL
LIN {X 0,Y 242.591,Z 511.375,A -85,B 0,C 180,E1 -19392.757,E2 -19392.757} C_VEL
LIN {X 0,Y 242.108,Z 509.982,A -85,B 0,C 180,E1 -19393.033,E2 -19393.033} C_VEL
LIN {X 0,Y 242.008,Z 509.447,A -85,B 0,C 180,E1 -19393.449,E2 -19393.449} C_VEL
LIN {X 0,Y 242.008,Z 509.46,A -85,B 0,C 180,E1 -19396.551,E2 -19396.551} C_VEL
LIN {X 0,Y 242.003,Z 509.454,A -85,B 0,C 180,E1 -19400.291,E2 -19400.291} C_VEL
LIN {X 0,Y 242.031,Z 509.442,A -85,B 0,C 180,E1 -19404.498,E2 -19404.498} C_VEL
LIN {X 0,Y 241.97,Z 509.448,A -85,B 0,C 180,E1 -19408.48,E2 -19408.48} C_VEL
LIN {X 0,Y 242.004,Z 509.466,A -85,B 0,C 180,E1 -19412.313,E2 -19412.313} C_VEL
LIN {X 0,Y 242.051,Z 509.429,A -85,B 0,C 180,E1 -19416.016,E2 -19416.016} C_VEL
LIN {X 0,Y 242.032,Z 509.46,A -85,B 0,C 180,E1 -19419.608,E2 -19419.608} C_VEL
LIN {X 0,Y 242.158,Z 509.414,A -85,B 0,C 180,E1 -19423.279,E2 -19423.279} C_VEL
LIN {X 0,Y 242.175,Z 509.421,A -85,B 0,C 180,E1 -19428.28,E2 -19428.28} C_VEL
LIN {X 0,Y 242.395,Z 509.389,A -85,B 0,C 180,E1 -19431.665,E2 -19431.665} C_VEL
LIN {X 0,Y 242.254,Z 509.426,A -85,B 0,C 180,E1 -19435.008,E2 -19435.008} C_VEL
LIN {X 0,Y 242.631,Z 509.346,A -85,B 0,C 180,E1 -19438.341,E2 -19438.341} C_VEL
LIN {X 0,Y 242.631,Z 509.383,A -85,B 0,C 180,E1 -19441.661,E2 -19441.661} C_VEL
LIN {X 0,Y 242.426,Z 509.376,A -85,B 0,C 180,E1 -19446.66,E2 -19446.66} C_VEL
LIN {X 0,Y 242.31,Z 509.428,A -85,B 0,C 180,E1 -19450.023,E2 -19450.023} C_VEL
LIN {X 0,Y 242.159,Z 509.421,A -85,B 0,C 180,E1 -19455.142,E2 -19455.142} C_VEL
LIN {X 0,Y 242.067,Z 509.444,A -85,B 0,C 180,E1 -19458.625,E2 -19458.625} C_VEL
LIN {X 0,Y 242.003,Z 509.444,A -85,B 0,C 180,E1 -19462.182,E2 -19462.182} C_VEL
LIN {X 0,Y 242.064,Z 509.438,A -85,B 0,C 180,E1 -19465.839,E2 -19465.839} C_VEL
LIN {X 0,Y 242.004,Z 509.461,A -85,B 0,C 180,E1 -19469.584,E2 -19469.584} C_VEL
LIN {X 0,Y 241.989,Z 509.445,A -85,B 0,C 180,E1 -19473.492,E2 -19473.492} C_VEL
LIN {X 0,Y 242.01,Z 509.449,A -85,B 0,C 180,E1 -19477.579,E2 -19477.579} C_VEL
LIN {X 0,Y 241.953,Z 509.461,A -85,B 0,C 180,E1 -19481.92,E2 -19481.92} C_VEL
LIN {X 0,Y 242.013,Z 509.65,A -85,B 0,C 180,E1 -19483.375,E2 -19483.375} C_VEL
LIN {X 0,Y 243.748,Z 516.362,A -85,B 0,C 180,E1 -19487.176,E2 -19487.176} C_VEL
LIN {X 0,Y 244.98,Z 519.122,A -85,B 0,C 180,E1 -19487.674,E2 -19487.674} C_VEL
LIN {X 0,Y 247.193,Z 522.717,A -85,B 0,C 180,E1 -19488.273,E2 -19488.273} C_VEL
LIN {X 0,Y 254.348,Z 535.887,A -85,B 0,C 180,E1 -19490.16,E2 -19490.16} C_VEL
LIN {X 0,Y 258.089,Z 543.305,A -85,B 0,C 180,E1 -19491.105,E2 -19491.105} C_VEL
LIN {X 0,Y 260.01,Z 550.51,A -85,B 0,C 180,E1 -19491.691,E2 -19491.691} C_VEL
LIN {X 0,Y 261.058,Z 558.135,A -85,B 0,C 180,E1 -19492.131,E2 -19492.131} C_VEL
LIN {X 0,Y 262.847,Z 573.625,A -85,B 0,C 180,E1 -19492.952,E2 -19492.952} C_VEL
LIN {X 0,Y 263.915,Z 580.965,A -85,B 0,C 180,E1 -19493.369,E2 -19493.369} C_VEL
LIN {X 0,Y 260.681,Z 651.939,A -85,B 0,C 180,E1 -19495.245,E2 -19495.245} C_VEL
LIN {X 0,Y 259.642,Z 663.64,A -85,B 0,C 180,E1 -19495.713,E2 -19495.713} C_VEL
LIN {X 0,Y 258.273,Z 674.628,A -85,B 0,C 180,E1 -19496.329,E2 -19496.329} C_VEL
LIN {X 0,Y 256.683,Z 684.418,A -85,B 0,C 180,E1 -19497.032,E2 -19497.032} C_VEL
LIN {X 0,Y 254.836,Z 694.386,A -85,B 0,C 180,E1 -19497.935,E2 -19497.935} C_VEL
LIN {X 0,Y 252.726,Z 704.303,A -85,B 0,C 180,E1 -19499.039,E2 -19499.039} C_VEL
LIN {X 0,Y 250.495,Z 713.664,A -85,B 0,C 180,E1 -19500.297,E2 -19500.297} C_VEL
LIN {X 0,Y 248.063,Z 723.447,A -85,B 0,C 180,E1 -19501.901,E2 -19501.901} C_VEL
LIN {X 0,Y 245.425,Z 732.464,A -85,B 0,C 180,E1 -19503.65,E2 -19503.65} C_VEL
LIN {X 0,Y 243.256,Z 739.435,A -85,B 0,C 180,E1 -19505.234,E2 -19505.234} C_VEL
LIN {X 0,Y 240.977,Z 746.959,A -85,B 0,C 180,E1 -19507.268,E2 -19507.268} C_VEL
LIN {X 0,Y 238.575,Z 754.571,A -85,B 0,C 180,E1 -19509.749,E2 -19509.749} C_VEL
LIN {X 0,Y 236.967,Z 759.937,A -85,B 0,C 180,E1 -19511.838,E2 -19511.838} C_VEL
LIN {X 0,Y 235.42,Z 765.413,A -85,B 0,C 180,E1 -19514.415,E2 -19514.415} C_VEL
LIN {X 0,Y 234.169,Z 769.86,A -85,B 0,C 180,E1 -19516.992,E2 -19516.992} C_VEL
LIN {X 0,Y 233.403,Z 773.411,A -85,B 0,C 180,E1 -19519.592,E2 -19519.592} C_VEL
LIN {X 0,Y 233.044,Z 775.355,A -85,B 0,C 180,E1 -19521.328,E2 -19521.328} C_VEL
LIN {X 0,Y 232.708,Z 778.286,A -85,B 0,C 180,E1 -19525.304,E2 -19525.304} C_VEL
LIN {X 0,Y 232.745,Z 779.347,A -85,B 0,C 180,E1 -19528.27,E2 -19528.27} C_VEL
LIN {X 0,Y 232.803,Z 779.602,A -85,B 0,C 180,E1 -19530,E2 -19530} C_VEL
LIN {X 0,Y 232.669,Z 778.869,A -85,B 0,C 180,E1 -19533.463,E2 -19533.463} C_VEL
LIN {X 0,Y 232.73,Z 778.049,A -85,B 0,C 180,E1 -19535.198,E2 -19535.198} C_VEL
LIN {X 0,Y 233.044,Z 775.355,A -85,B 0,C 180,E1 -19538.672,E2 -19538.672} C_VEL
LIN {X 0,Y 233.6,Z 772.393,A -85,B 0,C 180,E1 -19541.277,E2 -19541.277} C_VEL
LIN {X 0,Y 234.549,Z 768.562,A -85,B 0,C 180,E1 -19543.869,E2 -19543.869} C_VEL
LIN {X 0,Y 235.89,Z 763.796,A -85,B 0,C 180,E1 -19546.441,E2 -19546.441} C_VEL
LIN {X 0,Y 237.884,Z 756.847,A -85,B 0,C 180,E1 -19549.412,E2 -19549.412} C_VEL
LIN {X 0,Y 240.13,Z 749.634,A -85,B 0,C 180,E1 -19551.91,E2 -19551.91} C_VEL
LIN {X 0,Y 242.332,Z 742.56,A -85,B 0,C 180,E1 -19553.955,E2 -19553.955} C_VEL
LIN {X 0,Y 244.305,Z 736.099,A -85,B 0,C 180,E1 -19555.563,E2 -19555.563} C_VEL
LIN {X 0,Y 247.17,Z 726.625,A -85,B 0,C 180,E1 -19557.519,E2 -19557.519} C_VEL
LIN {X 0,Y 249.51,Z 718.025,A -85,B 0,C 180,E1 -19559.018,E2 -19559.018} C_VEL
LIN {X 0,Y 251.739,Z 708.697,A -85,B 0,C 180,E1 -19560.398,E2 -19560.398} C_VEL
LIN {X 0,Y 254.122,Z 697.893,A -85,B 0,C 180,E1 -19561.699,E2 -19561.699} C_VEL
LIN {X 0,Y 256.129,Z 687.637,A -85,B 0,C 180,E1 -19562.697,E2 -19562.697} C_VEL
LIN {X 0,Y 257.858,Z 677.347,A -85,B 0,C 180,E1 -19563.498,E2 -19563.498} C_VEL
LIN {X 0,Y 259.45,Z 665.464,A -85,B 0,C 180,E1 -19564.199,E2 -19564.199} C_VEL
LIN {X 0,Y 260.514,Z 653.906,A -85,B 0,C 180,E1 -19564.69,E2 -19564.69} C_VEL
LIN {X 0,Y 261.997,Z 625.398,A -85,B 0,C 180,E1 -19565.466,E2 -19565.466} C_VEL
LIN {X 0,Y 263.863,Z 579.626,A -85,B 0,C 180,E1 -19566.684,E2 -19566.684} C_VEL
LIN {X 0,Y 261.398,Z 566.172,A -85,B 0,C 180,E1 -19567.539,E2 -19567.539} C_VEL
LIN {X 0,Y 254.847,Z 550.759,A -85,B 0,C 180,E1 -19569.216,E2 -19569.216} C_VEL
LIN {X 0,Y 248.746,Z 538.295,A -85,B 0,C 180,E1 -19570.828,E2 -19570.828} C_VEL
LIN {X 0,Y 241.786,Z 525.502,A -85,B 0,C 180,E1 -19572.761,E2 -19572.761} C_VEL
LIN {X 0,Y 238.49,Z 520.125,A -85,B 0,C 180,E1 -19573.711,E2 -19573.711} C_VEL
LIN {X 0,Y 236.479,Z 516.25,A -85,B 0,C 180,E1 -19574.422,E2 -19574.422} C_VEL
LIN {X 0,Y 234.949,Z 510.417,A -85,B 0,C 180,E1 -19577.933,E2 -19577.933} C_VEL
LIN {X 0,Y 234.954,Z 510.331,A -85,B 0,C 180,E1 -19581.085,E2 -19581.085} C_VEL
LIN {X 0,Y 234.959,Z 510.33,A -85,B 0,C 180,E1 -19585.366,E2 -19585.366} C_VEL
LIN {X 0,Y 234.92,Z 510.347,A -85,B 0,C 180,E1 -19589.43,E2 -19589.43} C_VEL
LIN {X 0,Y 234.991,Z 510.314,A -85,B 0,C 180,E1 -19593.793,E2 -19593.793} C_VEL
LIN {X 0,Y 234.994,Z 510.306,A -85,B 0,C 180,E1 -19598.967,E2 -19598.967} C_VEL
LIN {X 0,Y 235.093,Z 510.327,A -85,B 0,C 180,E1 -19603.059,E2 -19603.059} C_VEL
LIN {X 0,Y 235.113,Z 510.294,A -85,B 0,C 180,E1 -19607.921,E2 -19607.921} C_VEL
LIN {X 0,Y 235.371,Z 510.284,A -85,B 0,C 180,E1 -19611.413,E2 -19611.413} C_VEL
LIN {X 0,Y 235.397,Z 510.252,A -85,B 0,C 180,E1 -19613.14,E2 -19613.14} C_VEL
LIN {X 0,Y 235.59,Z 510.26,A -85,B 0,C 180,E1 -19618.29,E2 -19618.29} C_VEL
LIN {X 0,Y 235.59,Z 510.222,A -85,B 0,C 180,E1 -19621.709,E2 -19621.709} C_VEL
LIN {X 0,Y 235.368,Z 510.285,A -85,B 0,C 180,E1 -19626.859,E2 -19626.859} C_VEL
LIN {X 0,Y 235.209,Z 510.273,A -85,B 0,C 180,E1 -19630.327,E2 -19630.327} C_VEL
LIN {X 0,Y 235.101,Z 510.305,A -85,B 0,C 180,E1 -19635.606,E2 -19635.606} C_VEL
LIN {X 0,Y 235.002,Z 510.317,A -85,B 0,C 180,E1 -19639.205,E2 -19639.205} C_VEL
LIN {X 0,Y 234.955,Z 510.321,A -85,B 0,C 180,E1 -19642.882,E2 -19642.882} C_VEL
LIN {X 0,Y 234.965,Z 510.335,A -85,B 0,C 180,E1 -19646.657,E2 -19646.657} C_VEL
LIN {X 0,Y 234.927,Z 510.32,A -85,B 0,C 180,E1 -19650.567,E2 -19650.567} C_VEL
LIN {X 0,Y 234.955,Z 510.33,A -85,B 0,C 180,E1 -19654.633,E2 -19654.633} C_VEL
LIN {X 0,Y 234.962,Z 510.34,A -85,B 0,C 180,E1 -19658.952,E2 -19658.952} C_VEL
LIN {X 0,Y 234.982,Z 510.332,A -85,B 0,C 180,E1 -19663.463,E2 -19663.463} C_VEL
LIN {X 0,Y 234.982,Z 510.581,A -85,B 0,C 180,E1 -19665.213,E2 -19665.213} C_VEL
LIN {X 0,Y 235.27,Z 511.682,A -85,B 0,C 180,E1 -19665.56,E2 -19665.56} C_VEL
LIN {X 0,Y 236.918,Z 514.378,A -85,B 0,C 180,E1 -19666.082,E2 -19666.082} C_VEL
LIN {X 0,Y 238.285,Z 515.966,A -85,B 0,C 180,E1 -19666.464,E2 -19666.464} C_VEL
LIN {X 0,Y 240.44,Z 519.15,A -85,B 0,C 180,E1 -19667.081,E2 -19667.081} C_VEL
LIN {X 0,Y 248.763,Z 531.947,A -85,B 0,C 180,E1 -19669.331,E2 -19669.331} C_VEL
LIN {X 0,Y 262.368,Z 554.496,A -85,B 0,C 180,E1 -19672.621,E2 -19672.621} C_VEL
LIN {X 0,Y 269.372,Z 563.685,A -85,B 0,C 180,E1 -19674.057,E2 -19674.057} C_VEL
LIN {X 0,Y 279.851,Z 575.487,A -85,B 0,C 180,E1 -19675.968,E2 -19675.968} C_VEL
LIN {X 0,Y 295.828,Z 590.584,A -85,B 0,C 180,E1 -19678.532,E2 -19678.532} C_VEL
LIN {X 0,Y 305,Z 598.699,A -85,B 0,C 180,E1 -19680.146,E2 -19680.146} C_VEL
LIN {X 0,Y 313.689,Z 606.175,A -85,B 0,C 180,E1 -19681.877,E2 -19681.877} C_VEL
LIN {X 0,Y 322.309,Z 613.401,A -85,B 0,C 180,E1 -19683.829,E2 -19683.829} C_VEL
LIN {X 0,Y 329.59,Z 619.301,A -85,B 0,C 180,E1 -19685.633,E2 -19685.633} C_VEL
LIN {X 0,Y 336.528,Z 624.595,A -85,B 0,C 180,E1 -19687.475,E2 -19687.475} C_VEL
LIN {X 0,Y 343.685,Z 630.293,A -85,B 0,C 180,E1 -19689.57,E2 -19689.57} C_VEL
LIN {X 0,Y 350.315,Z 634.945,A -85,B 0,C 180,E1 -19691.7,E2 -19691.7} C_VEL
LIN {X 0,Y 355.267,Z 638.899,A -85,B 0,C 180,E1 -19693.495,E2 -19693.495} C_VEL
LIN {X 0,Y 359.789,Z 641.813,A -85,B 0,C 180,E1 -19695.29,E2 -19695.29} C_VEL
LIN {X 0,Y 363.33,Z 643.906,A -85,B 0,C 180,E1 -19696.847,E2 -19696.847} C_VEL
LIN {X 0,Y 367.378,Z 647.248,A -85,B 0,C 180,E1 -19698.972,E2 -19698.972} C_VEL
LIN {X 0,Y 370.781,Z 649.415,A -85,B 0,C 180,E1 -19701.09,E2 -19701.09} C_VEL
LIN {X 0,Y 373.533,Z 650.884,A -85,B 0,C 180,E1 -19703.249,E2 -19703.249} C_VEL
LIN {X 0,Y 375.464,Z 651.762,A -85,B 0,C 180,E1 -19705.306,E2 -19705.306} C_VEL
LIN {X 0,Y 376.675,Z 652.212,A -85,B 0,C 180,E1 -19707.327,E2 -19707.327} C_VEL
LIN {X 0,Y 377.186,Z 652.514,A -85,B 0,C 180,E1 -19708.932,E2 -19708.932} C_VEL
LIN {X 0,Y 377.302,Z 652.399,A -85,B 0,C 180,E1 -19710,E2 -19710} C_VEL
LIN {X 0,Y 377.186,Z 652.52,A -85,B 0,C 180,E1 -19711.068,E2 -19711.068} C_VEL
LIN {X 0,Y 376.429,Z 652.081,A -85,B 0,C 180,E1 -19713.211,E2 -19713.211} C_VEL
LIN {X 0,Y 374.871,Z 651.568,A -85,B 0,C 180,E1 -19715.379,E2 -19715.379} C_VEL
LIN {X 0,Y 372.525,Z 650.431,A -85,B 0,C 180,E1 -19717.589,E2 -19717.589} C_VEL
LIN {X 0,Y 369.326,Z 648.56,A -85,B 0,C 180,E1 -19719.861,E2 -19719.861} C_VEL
LIN {X 0,Y 366.079,Z 646.213,A -85,B 0,C 180,E1 -19721.739,E2 -19721.739} C_VEL
LIN {X 0,Y 361.706,Z 642.827,A -85,B 0,C 180,E1 -19723.895,E2 -19723.895} C_VEL
LIN {X 0,Y 356.889,Z 639.971,A -85,B 0,C 180,E1 -19725.892,E2 -19725.892} C_VEL
LIN {X 0,Y 351.85,Z 636.238,A -85,B 0,C 180,E1 -19727.766,E2 -19727.766} C_VEL
LIN {X 0,Y 347.36,Z 632.8,A -85,B 0,C 180,E1 -19729.284,E2 -19729.284} C_VEL
LIN {X 0,Y 341.665,Z 628.766,A -85,B 0,C 180,E1 -19731.043,E2 -19731.043} C_VEL
